C07281=1059.904,-11.969,431.979,171.523,28.026,155.225
C07282=1059.910,-11.719,431.964,171.524,28.029,155.225
C07283=1059.916,-11.470,431.951,171.526,28.031,155.225
C07284=1059.922,-11.220,431.937,171.528,28.033,155.226
C07285=1059.928,-10.971,431.922,171.529,28.035,155.226
C07286=1059.934,-10.722,431.909,171.531,28.038,155.226
C07287=1059.941,-10.472,431.894,171.532,28.040,155.226
C07288=1059.946,-10.222,431.880,171.534,28.042,155.227
C07289=1059.953,-9.972,431.867,171.536,28.045,155.227
C07290=1059.959,-9.723,431.852,171.537,28.047,155.227
C07291=1059.965,-9.473,431.838,171.539,28.049,155.228
C07292=1059.972,-9.225,431.824,171.540,28.051,155.228
C07293=1059.977,-8.975,431.810,171.541,28.054,155.228
C07294=1059.983,-8.725,431.796,171.543,28.056,155.228
C07295=1059.990,-8.476,431.782,171.545,28.058,155.229
C07296=1059.996,-8.226,431.767,171.546,28.060,155.229
C07297=1060.001,-7.977,431.753,171.548,28.063,155.229
C07298=1060.008,-7.727,431.739,171.549,28.065,155.230
C07299=1060.014,-7.478,431.725,171.551,28.067,155.230
C07300=1060.020,-7.228,431.710,171.553,28.069,155.230
C07301=1060.027,-6.979,431.696,171.554,28.072,155.230
C07302=1060.033,-6.729,431.682,171.556,28.074,155.231
C07303=1060.039,-6.480,431.668,171.557,28.076,155.231
C07304=1060.045,-6.229,431.653,171.558,28.079,155.231
C07305=1060.051,-5.981,431.639,171.560,28.081,155.232
C07306=1060.057,-5.731,431.625,171.562,28.083,155.232
C07307=1060.063,-5.482,431.611,171.563,28.085,155.232
C07308=1060.070,-5.232,431.597,171.565,28.088,155.232
C07309=1060.076,-4.983,431.582,171.566,28.090,155.233
C07310=1060.082,-4.732,431.568,171.568,28.092,155.233
C07311=1060.088,-4.484,431.554,171.570,28.094,155.233
C07312=1060.095,-4.234,431.539,171.571,28.097,155.233
C07313=1060.101,-3.984,431.525,171.573,28.099,155.234
C07314=1060.106,-3.735,431.510,171.574,28.101,155.234
C07315=1060.113,-3.485,431.497,171.575,28.104,155.234
C07316=1060.119,-3.236,431.482,171.577,28.106,155.235
C07317=1060.125,-2.986,431.467,171.579,28.108,155.235
C07318=1060.131,-2.737,431.453,171.580,28.110,155.235
C07319=1060.137,-2.455,431.437,171.582,28.113,155.236
C07320=1060.145,-2.174,431.420,171.583,28.116,155.236
C07321=1060.151,-1.893,431.404,171.585,28.118,155.236
C07322=1060.158,-1.612,431.388,171.587,28.121,155.237
C07323=1060.164,-1.362,431.373,171.588,28.123,155.237
C07324=1060.170,-1.113,431.359,171.590,28.126,155.237
C07325=1060.176,-0.863,431.344,171.591,28.128,155.238
C07326=1060.182,-0.614,431.330,171.593,28.131,155.238
C07327=1060.188,-0.364,431.315,171.595,28.134,155.238
C07328=1060.194,-0.114,431.301,171.596,28.136,155.239
C07329=1060.200,0.135,431.286,171.598,28.138,155.239
C07330=1060.207,0.385,431.271,171.600,28.140,155.239
C07331=1060.212,0.634,431.257,171.600,28.143,155.239
C07332=1060.218,0.884,431.242,171.602,28.145,155.240
C07333=1060.224,1.133,431.228,171.603,28.147,155.240
C07334=1060.231,1.383,431.213,171.605,28.150,155.240
C07335=1060.236,1.632,431.198,171.607,28.152,155.241
C07336=1060.243,1.882,431.184,171.608,28.155,155.241
C07337=1060.248,2.131,431.169,171.610,28.157,155.241
C07338=1060.254,2.381,431.154,171.612,28.160,155.242
C07339=1060.260,2.630,431.139,171.612,28.162,155.242
C07340=1060.266,2.879,431.124,171.614,28.164,155.242
C07341=1060.272,3.130,431.110,171.615,28.166,155.242
C07342=1060.278,3.379,431.096,171.617,28.169,155.243
C07343=1060.284,3.628,431.081,171.619,28.171,155.243
C07344=1060.291,3.878,431.066,171.620,28.173,155.243
C07345=1060.297,4.127,431.051,171.622,28.176,155.244
C07346=1060.303,4.377,431.036,171.624,28.179,155.244
C07347=1060.309,4.626,431.021,171.625,28.181,155.244
C07348=1060.315,4.876,431.007,171.626,28.183,155.245
C07349=1060.321,5.125,430.992,171.627,28.186,155.245
C07350=1060.327,5.374,430.978,171.629,28.188,155.245
C07351=1060.333,5.624,430.963,171.631,28.190,155.246
C07352=1060.340,5.874,430.948,171.632,28.193,155.246
C07353=1060.345,6.123,430.933,171.634,28.195,155.246
C07354=1060.352,6.372,430.918,171.636,28.197,155.246
C07355=1060.358,6.622,430.903,171.637,28.200,155.247
C07356=1060.364,6.871,430.889,171.638,28.202,155.247
C07357=1060.370,7.121,430.873,171.640,28.204,155.247
C07358=1060.376,7.371,430.858,171.641,28.207,155.248
C07359=1060.382,7.620,430.844,171.643,28.209,155.248
C07360=1060.388,7.870,430.830,171.644,28.212,155.248
C07361=1060.394,8.119,430.815,171.646,28.214,155.249
C07362=1060.400,8.368,430.800,171.648,28.217,155.249
C07363=1060.406,8.618,430.785,171.648,28.219,155.249
C07364=1060.413,8.868,430.770,171.650,28.221,155.250
C07365=1060.419,9.117,430.755,171.652,28.224,155.250
C07366=1060.425,9.366,430.741,171.653,28.226,155.250
C07367=1060.431,9.616,430.726,171.655,28.228,155.251
C07368=1060.438,9.866,430.711,171.656,28.231,155.251
C07369=1060.444,10.115,430.694,171.658,28.233,155.251
C07370=1060.450,10.364,430.680,171.660,28.236,155.251
C07371=1060.456,10.614,430.665,171.660,28.238,155.252
C07372=1060.462,10.863,430.650,171.662,28.240,155.252
C07373=1060.468,11.112,430.635,171.664,28.243,155.252
C07374=1060.474,11.362,430.620,171.665,28.245,155.253
C07375=1060.481,11.612,430.605,171.667,28.248,155.253
C07376=1060.487,11.861,430.591,171.669,28.250,155.253
C07377=1060.493,12.111,430.575,171.670,28.252,155.254
C07378=1060.499,12.360,430.560,171.671,28.255,155.254
C07379=1060.505,12.610,430.545,171.672,28.257,155.254
C07380=1060.511,12.859,430.531,171.674,28.259,155.255
C07381=1060.518,13.109,430.515,171.676,28.262,155.255
C07382=1060.524,13.357,430.500,171.677,28.264,155.255
C07383=1060.531,13.642,430.483,171.679,28.267,155.256
C07384=1060.538,13.925,430.466,171.681,28.269,155.256
C07385=1060.546,14.208,430.449,171.682,28.272,155.256
C07386=1060.552,14.491,430.432,171.684,28.275,155.257
C07387=1060.559,14.740,430.416,171.685,28.277,155.257
C07388=1060.564,14.990,430.401,171.687,28.280,155.257
C07389=1060.570,15.239,430.386,171.689,28.282,155.258
C07390=1060.576,15.489,430.371,171.690,28.285,155.258
C07391=1060.582,15.739,430.356,171.692,28.287,155.258
C07392=1060.588,15.987,430.340,171.693,28.290,155.259
C07393=1060.595,16.237,430.325,171.694,28.292,155.259
C07394=1060.600,16.487,430.310,171.696,28.295,155.259
C07395=1060.607,16.737,430.295,171.697,28.297,155.260
C07396=1060.613,16.986,430.279,171.699,28.299,155.260
C07397=1060.618,17.235,430.264,171.701,28.302,155.260
C07398=1060.625,17.485,430.249,171.702,28.304,155.261
C07399=1060.631,17.734,430.234,171.703,28.307,155.261
C07400=1060.637,17.984,430.218,171.705,28.309,155.261
C07401=1060.643,18.233,430.203,171.706,28.312,155.262
C07402=1060.648,18.483,430.188,171.708,28.314,155.262
C07403=1060.655,18.732,430.172,171.709,28.317,155.262
C07404=1060.662,18.981,430.157,171.711,28.319,155.263
C07405=1060.667,19.231,430.142,171.713,28.321,155.263
C07406=1060.674,19.480,430.126,171.713,28.324,155.263
C07407=1060.680,19.730,430.111,171.715,28.326,155.264
C07408=1060.685,19.979,430.096,171.716,28.329,155.264
C07409=1060.692,20.228,430.080,171.718,28.331,155.264
C07410=1060.698,20.478,430.065,171.720,28.334,155.265
C07411=1060.704,20.728,430.050,171.721,28.336,155.265
C07412=1060.710,20.977,430.033,171.722,28.339,155.265
C07413=1060.716,21.227,430.019,171.724,28.341,155.266
C07414=1060.722,21.476,430.002,171.725,28.344,155.266
C07415=1060.728,21.725,429.988,171.727,28.346,155.266
C07416=1060.734,21.974,429.971,171.728,28.349,155.267
C07417=1060.740,22.224,429.956,171.730,28.351,155.267
C07418=1060.746,22.474,429.941,171.732,28.354,155.267
C07419=1060.753,22.723,429.925,171.732,28.356,155.268
C07420=1060.758,22.973,429.910,171.734,28.359,155.268
C07421=1060.765,23.222,429.894,171.736,28.361,155.268
C07422=1060.770,23.471,429.879,171.737,28.364,155.269
C07423=1060.777,23.720,429.863,171.739,28.366,155.269
C07424=1060.782,23.970,429.848,171.741,28.369,155.269
C07425=1060.789,24.219,429.832,171.741,28.371,155.270
C07426=1060.795,24.469,429.816,171.743,28.374,155.270
C07427=1060.801,24.718,429.801,171.744,28.376,155.270
C07428=1060.807,24.968,429.785,171.746,28.379,155.271
C07429=1060.814,25.217,429.770,171.748,28.381,155.271
C07430=1060.819,25.467,429.754,171.749,28.384,155.271
C07431=1060.825,25.717,429.738,171.750,28.386,155.272
C07432=1060.831,25.966,429.723,171.752,28.388,155.272
C07433=1060.837,26.215,429.707,171.753,28.391,155.272
C07434=1060.844,26.465,429.692,171.755,28.393,155.273
C07435=1060.849,26.714,429.676,171.756,28.396,155.273
C07436=1060.856,26.963,429.660,171.758,28.398,155.273
C07437=1060.862,27.213,429.645,171.759,28.400,155.274
C07438=1060.868,27.462,429.628,171.760,28.403,155.274
C07439=1060.874,27.712,429.613,171.762,28.406,155.275
C07440=1060.880,27.961,429.597,171.764,28.408,155.275
C07441=1060.887,28.210,429.581,171.765,28.411,155.275
C07442=1060.892,28.460,429.566,171.767,28.413,155.275
C07443=1060.898,28.710,429.550,171.768,28.416,155.276
C07444=1060.905,28.959,429.534,171.769,28.418,155.276
C07445=1060.911,29.209,429.518,171.771,28.421,155.277
C07446=1060.917,29.458,429.502,171.772,28.423,155.277
C07447=1060.924,29.743,429.485,171.774,28.426,155.277
C07448=1060.930,30.027,429.466,171.776,28.429,155.278
C07449=1060.938,30.312,429.449,171.777,28.432,155.278
C07450=1060.944,30.596,429.430,171.779,28.435,155.279
C07451=1060.950,30.846,429.414,171.780,28.438,155.279
C07452=1060.956,31.096,429.398,171.782,28.440,155.279
C07453=1060.962,31.345,429.383,171.784,28.443,155.280
C07454=1060.968,31.594,429.366,171.785,28.445,155.280
C07455=1060.974,31.844,429.351,171.786,28.447,155.280
C07456=1060.980,32.093,429.334,171.787,28.450,155.281
C07457=1060.987,32.342,429.319,171.789,28.452,155.281
C07458=1060.993,32.592,429.303,171.791,28.455,155.281
C07459=1060.998,32.842,429.287,171.792,28.458,155.282
C07460=1061.004,33.091,429.271,171.794,28.460,155.282
C07461=1061.011,33.340,429.255,171.795,28.463,155.282
C07462=1061.017,33.589,429.239,171.796,28.465,155.283
C07463=1061.023,33.839,429.223,171.798,28.468,155.283
C07464=1061.028,34.089,429.207,171.799,28.470,155.283
C07465=1061.035,34.338,429.191,171.801,28.473,155.284
C07466=1061.041,34.587,429.175,171.803,28.476,155.284
C07467=1061.047,34.836,429.159,171.803,28.478,155.284
C07468=1061.053,35.086,429.143,171.805,28.480,155.285
C07469=1061.059,35.335,429.126,171.807,28.483,155.285
C07470=1061.065,35.585,429.111,171.808,28.485,155.286
C07471=1061.071,35.834,429.095,171.810,28.488,155.286
C07472=1061.077,36.083,429.079,171.812,28.490,155.286
C07473=1061.083,36.333,429.063,171.812,28.493,155.287
C07474=1061.089,36.582,429.046,171.814,28.495,155.287
C07475=1061.096,36.831,429.031,171.815,28.498,155.287
C07476=1061.102,37.081,429.014,171.817,28.501,155.288
C07477=1061.108,37.331,428.998,171.819,28.503,155.288
C07478=1061.114,37.580,428.982,171.820,28.506,155.288
C07479=1061.120,37.829,428.965,171.821,28.508,155.289
C07480=1061.126,38.079,428.950,171.823,28.511,155.289
C07481=1061.132,38.329,428.934,171.824,28.513,155.289
C07482=1061.138,38.578,428.917,171.826,28.516,155.290
C07483=1061.144,38.827,428.901,171.827,28.518,155.290
C07484=1061.150,39.077,428.885,171.828,28.521,155.291
C07485=1061.156,39.326,428.868,171.830,28.523,155.291
C07486=1061.162,39.575,428.852,171.831,28.526,155.291
C07487=1061.168,39.825,428.836,171.833,28.529,155.292
C07488=1061.173,40.074,428.820,171.835,28.532,155.292
C07489=1061.179,40.323,428.803,171.836,28.534,155.292
C07490=1061.185,40.573,428.787,171.837,28.536,155.293
C07491=1061.192,40.823,428.771,171.838,28.539,155.293
C07492=1061.198,41.072,428.754,171.840,28.541,155.293
C07493=1061.204,41.321,428.737,171.842,28.544,155.294
C07494=1061.210,41.570,428.721,171.843,28.547,155.294
C07495=1061.216,41.820,428.705,171.844,28.549,155.294
C07496=1061.222,42.069,428.689,171.846,28.552,155.295
C07497=1061.228,42.318,428.672,171.847,28.555,155.295
C07498=1061.234,42.568,428.656,171.849,28.557,155.296
C07499=1061.240,42.817,428.640,171.851,28.560,155.296
C07500=1061.246,43.067,428.623,171.852,28.562,155.296
C07501=1061.252,43.316,428.607,171.853,28.564,155.297
C07502=1061.258,43.566,428.591,171.854,28.567,155.297
C07503=1061.264,43.815,428.574,171.856,28.570,155.297
C07504=1061.270,44.064,428.557,171.858,28.573,155.298
C07505=1061.276,44.313,428.541,171.859,28.575,155.298
C07506=1061.282,44.563,428.524,171.860,28.577,155.299
C07507=1061.288,44.812,428.508,171.862,28.580,155.299
C07508=1061.294,45.062,428.491,171.863,28.583,155.299
C07509=1061.300,45.312,428.475,171.865,28.586,155.300
C07510=1061.306,45.561,428.458,171.866,28.588,155.300
C07511=1061.312,45.845,428.439,171.868,28.591,155.300
C07512=1061.319,46.130,428.420,171.870,28.594,155.301
C07513=1061.326,46.414,428.401,171.871,28.597,155.301
C07514=1061.333,46.699,428.382,171.873,28.600,155.302
C07515=1061.339,46.948,428.366,171.874,28.603,155.302
C07516=1061.344,47.198,428.349,171.876,28.605,155.302
C07517=1061.350,47.447,428.332,171.877,28.608,155.303
C07518=1061.356,47.696,428.316,171.878,28.611,155.303
C07519=1061.362,47.946,428.299,171.880,28.613,155.304
C07520=1061.368,48.196,428.283,171.881,28.616,155.304
C07521=1061.374,48.444,428.266,171.883,28.618,155.304
C07522=1061.380,48.694,428.249,171.885,28.621,155.305
C07523=1061.385,48.943,428.233,171.885,28.624,155.305
C07524=1061.392,49.192,428.216,171.887,28.627,155.306
C07525=1061.398,49.442,428.199,171.889,28.629,155.306
C07526=1061.404,49.691,428.183,171.890,28.632,155.306
C07527=1061.410,49.940,428.165,171.892,28.634,155.307
C07528=1061.416,50.190,428.149,171.892,28.637,155.307
C07529=1061.422,50.439,428.133,171.894,28.639,155.307
C07530=1061.428,50.689,428.115,171.896,28.642,155.308
C07531=1061.434,50.938,428.098,171.897,28.645,155.308
C07532=1061.440,51.188,428.082,171.899,28.647,155.309
C07533=1061.445,51.437,428.065,171.900,28.650,155.309
C07534=1061.452,51.687,428.048,171.901,28.652,155.309
C07535=1061.458,51.935,428.031,171.903,28.655,155.310
C07536=1061.464,52.185,428.015,171.905,28.658,155.310
C07537=1061.469,52.434,427.998,171.906,28.661,155.310
C07538=1061.475,52.683,427.981,171.908,28.663,155.311
C07539=1061.482,52.933,427.964,171.908,28.665,155.311
C07540=1061.487,53.182,427.947,171.910,28.668,155.311
C07541=1061.493,53.432,427.930,171.912,28.671,155.312
C07542=1061.500,53.681,427.913,171.913,28.673,155.312
C07543=1061.505,53.931,427.896,171.915,28.676,155.313
C07544=1061.512,54.179,427.879,171.916,28.678,155.313
C07545=1061.518,54.429,427.863,171.917,28.681,155.313
C07546=1061.523,54.679,427.846,171.919,28.683,155.314
C07547=1061.530,54.928,427.829,171.921,28.686,155.314
C07548=1061.536,55.177,427.813,171.922,28.689,155.314
C07549=1061.542,55.427,427.795,171.924,28.692,155.315
C07550=1061.548,55.676,427.778,171.924,28.694,155.315
C07551=1061.554,55.925,427.761,171.926,28.697,155.316
C07552=1061.560,56.174,427.744,171.928,28.699,155.316
C07553=1061.566,56.424,427.727,171.929,28.702,155.316
C07554=1061.572,56.673,427.710,171.931,28.704,155.317
C07555=1061.578,56.923,427.693,171.932,28.707,155.317
C07556=1061.584,57.172,427.676,171.933,28.710,155.317
C07557=1061.590,57.421,427.660,171.935,28.712,155.318
C07558=1061.596,57.670,427.642,171.937,28.715,155.318
C07559=1061.602,57.920,427.626,171.938,28.717,155.319
C07560=1061.608,58.169,427.608,171.940,28.720,155.319
C07561=1061.614,58.418,427.591,171.940,28.723,155.319
C07562=1061.621,58.668,427.574,171.942,28.725,155.320
C07563=1061.626,58.917,427.557,171.944,28.728,155.320
C07564=1061.633,59.167,427.540,171.945,28.730,155.320
C07565=1061.639,59.416,427.523,171.947,28.733,155.321
C07566=1061.645,59.665,427.506,171.948,28.735,155.321
C07567=1061.651,59.915,427.489,171.949,28.738,155.322
C07568=1061.657,60.164,427.472,171.951,28.741,155.322
C07569=1061.664,60.414,427.454,171.953,28.743,155.322
C07570=1061.669,60.663,427.438,171.954,28.746,155.323
C07571=1061.675,60.912,427.420,171.956,28.748,155.323
C07572=1061.682,61.161,427.403,171.957,28.750,155.323
C07573=1061.688,61.411,427.387,171.958,28.753,155.324
C07574=1061.694,61.660,427.369,171.960,28.756,155.324
C07575=1061.701,61.944,427.350,171.961,28.759,155.324
C07576=1061.708,62.228,427.330,171.963,28.762,155.325
C07577=1061.715,62.514,427.310,171.965,28.765,155.325
C07578=1061.721,62.797,427.291,171.966,28.768,155.326
C07579=1061.728,63.047,427.274,171.968,28.770,155.326
C07580=1061.734,63.296,427.256,171.970,28.773,155.326
C07581=1061.740,63.546,427.239,171.971,28.775,155.327
C07582=1061.747,63.794,427.222,171.973,28.778,155.327
C07583=1061.753,64.044,427.204,171.974,28.780,155.328
C07584=1061.759,64.293,427.188,171.975,28.783,155.328
C07585=1061.765,64.543,427.170,171.977,28.786,155.328
C07586=1061.770,64.792,427.153,171.978,28.788,155.329
C07587=1061.776,65.041,427.136,171.980,28.791,155.329
C07588=1061.783,65.291,427.118,171.982,28.793,155.329
C07589=1061.789,65.539,427.101,171.982,28.796,155.330
C07590=1061.795,65.789,427.083,171.984,28.799,155.330
C07591=1061.800,66.039,427.066,171.986,28.802,155.331
C07592=1061.807,66.288,427.049,171.987,28.804,155.331
C07593=1061.813,66.537,427.031,171.989,28.806,155.331
C07594=1061.818,66.786,427.014,171.991,28.809,155.332
C07595=1061.825,67.036,426.996,171.991,28.812,155.332
C07596=1061.830,67.285,426.979,171.993,28.815,155.333
C07597=1061.837,67.535,426.961,171.994,28.817,155.333
C07598=1061.843,67.783,426.944,171.996,28.820,155.333
C07599=1061.849,68.033,426.926,171.998,28.822,155.334
C07600=1061.854,68.283,426.909,171.999,28.825,155.334
C07601=1061.860,68.532,426.891,172.000,28.828,155.334
C07602=1061.867,68.781,426.874,172.002,28.830,155.335
C07603=1061.873,69.031,426.856,172.003,28.833,155.335
C07604=1061.878,69.280,426.839,172.005,28.835,155.336
C07605=1061.885,69.529,426.821,172.007,28.838,155.336
C07606=1061.891,69.778,426.804,172.007,28.841,155.336
C07607=1061.897,70.028,426.786,172.009,28.843,155.337
C07608=1061.902,70.277,426.768,172.010,28.846,155.337
C07609=1061.908,70.526,426.751,172.012,28.848,155.337
C07610=1061.915,70.776,426.733,172.014,28.851,155.338
C07611=1061.920,71.025,426.716,172.015,28.854,155.338
C07612=1061.926,71.274,426.698,172.016,28.856,155.339
C07613=1061.932,71.523,426.680,172.018,28.859,155.339
C07614=1061.938,71.773,426.662,172.019,28.862,155.339
C07615=1061.944,72.022,426.645,172.021,28.865,155.340
C07616=1061.950,72.272,426.627,172.023,28.867,155.340
C07617=1061.956,72.520,426.609,172.024,28.870,155.341
C07618=1061.962,72.770,426.591,172.025,28.872,155.341
C07619=1061.968,73.019,426.574,172.027,28.875,155.341
C07620=1061.974,73.269,426.556,172.028,28.878,155.342
C07621=1061.979,73.518,426.538,172.030,28.881,155.342
C07622=1061.986,73.767,426.521,172.031,28.883,155.343
C07623=1061.992,74.016,426.503,172.032,28.886,155.343
C07624=1061.998,74.266,426.485,172.034,28.888,155.343
C07625=1062.004,74.516,426.467,172.035,28.891,155.344
C07626=1062.010,74.764,426.449,172.037,28.894,155.344
C07627=1062.016,75.014,426.431,172.039,28.896,155.344
C07628=1062.021,75.263,426.414,172.040,28.899,155.345
C07629=1062.028,75.513,426.396,172.041,28.902,155.345
C07630=1062.034,75.761,426.379,172.043,28.904,155.346
C07631=1062.040,76.011,426.361,172.044,28.907,155.346
C07632=1062.046,76.259,426.342,172.046,28.909,155.346
C07633=1062.052,76.509,426.324,172.048,28.912,155.347
C07634=1062.058,76.759,426.307,172.049,28.915,155.347
C07635=1062.064,77.008,426.289,172.050,28.917,155.348
C07636=1062.070,77.258,426.271,172.052,28.920,155.348
C07637=1062.075,77.506,426.253,172.053,28.922,155.348
C07638=1062.082,77.756,426.235,172.055,28.925,155.349
C07639=1062.088,78.040,426.215,172.056,28.928,155.349
C07640=1062.096,78.324,426.194,172.058,28.931,155.350
C07641=1062.102,78.608,426.174,172.060,28.934,155.350
C07642=1062.109,78.892,426.153,172.061,28.937,155.351
C07643=1062.115,79.142,426.135,172.063,28.940,155.351
C07644=1062.121,79.391,426.118,172.065,28.943,155.351
C07645=1062.126,79.641,426.099,172.066,28.946,155.352
C07646=1062.132,79.890,426.080,172.068,28.948,155.352
C07647=1062.138,80.139,426.063,172.068,28.951,155.353
C07648=1062.144,80.389,426.045,172.070,28.953,155.353
C07649=1062.150,80.637,426.027,172.072,28.956,155.353
C07650=1062.156,80.887,426.009,172.073,28.959,155.354
C07651=1062.162,81.135,425.990,172.075,28.961,155.354
C07652=1062.168,81.385,425.973,172.077,28.964,155.354
C07653=1062.173,81.635,425.954,172.077,28.967,155.355
C07654=1062.179,81.884,425.936,172.079,28.969,155.355
C07655=1062.185,82.133,425.918,172.081,28.972,155.356
C07656=1062.191,82.383,425.900,172.082,28.975,155.356
C07657=1062.197,82.631,425.882,172.084,28.978,155.356
C07658=1062.203,82.881,425.864,172.086,28.980,155.357
C07659=1062.209,83.130,425.845,172.086,28.983,155.357
C07660=1062.215,83.380,425.827,172.088,28.985,155.358
C07661=1062.221,83.629,425.808,172.090,28.988,155.358
C07662=1062.227,83.878,425.791,172.091,28.991,155.358
C07663=1062.233,84.128,425.773,172.093,28.993,155.359
C07664=1062.239,84.377,425.754,172.095,28.996,155.359
C07665=1062.245,84.626,425.736,172.095,28.999,155.360
C07666=1062.250,84.875,425.717,172.097,29.001,155.360
C07667=1062.256,85.125,425.699,172.098,29.004,155.360
C07668=1062.262,85.373,425.681,172.100,29.007,155.361
C07669=1062.268,85.623,425.663,172.102,29.009,155.361
C07670=1062.275,85.872,425.644,172.103,29.012,155.361
C07671=1062.280,86.121,425.627,172.105,29.015,155.362
C07672=1062.286,86.371,425.608,172.106,29.017,155.362
C07673=1062.292,86.620,425.590,172.107,29.020,155.363
C07674=1062.299,86.870,425.571,172.109,29.023,155.363
C07675=1062.304,87.118,425.553,172.111,29.025,155.364
C07676=1062.310,87.368,425.535,172.112,29.028,155.364
C07677=1062.317,87.617,425.516,172.114,29.030,155.364
C07678=1062.322,87.866,425.498,172.116,29.033,155.365
C07679=1062.328,88.115,425.479,172.116,29.036,155.365
C07680=1062.334,88.365,425.461,172.118,29.038,155.365
C07681=1062.341,88.614,425.443,172.120,29.041,155.366
C07682=1062.346,88.863,425.425,172.121,29.044,155.366
C07683=1062.352,89.113,425.406,172.123,29.047,155.367
C07684=1062.358,89.362,425.387,172.125,29.049,155.367
C07685=1062.365,89.611,425.369,172.125,29.051,155.367
C07686=1062.370,89.860,425.351,172.127,29.054,155.368
C07687=1062.376,90.109,425.332,172.129,29.057,155.368
C07688=1062.382,90.358,425.313,172.130,29.060,155.369
C07689=1062.388,90.608,425.295,172.132,29.062,155.369
C07690=1062.394,90.857,425.277,172.134,29.065,155.369
C07691=1062.400,91.106,425.258,172.135,29.068,155.370
C07692=1062.406,91.356,425.240,172.136,29.070,155.370
C07693=1062.412,91.605,425.221,172.138,29.073,155.371
C07694=1062.418,91.854,425.202,172.139,29.076,155.371
C07695=1062.424,92.103,425.184,172.141,29.078,155.371
C07696=1062.429,92.353,425.165,172.143,29.081,155.372
C07697=1062.436,92.602,425.146,172.144,29.084,155.372
C07698=1062.441,92.851,425.128,172.146,29.086,155.372
C07699=1062.447,93.100,425.110,172.147,29.089,155.373
C07700=1062.453,93.350,425.090,172.148,29.092,155.373
C07701=1062.459,93.599,425.072,172.150,29.094,155.374
C07702=1062.464,93.848,425.053,172.151,29.097,155.374
C07703=1062.471,94.132,425.032,172.153,29.100,155.375
C07704=1062.479,94.416,425.011,172.155,29.103,155.375
C07705=1062.485,94.701,424.989,172.156,29.107,155.376
C07706=1062.492,94.985,424.968,172.158,29.109,155.376
C07707=1062.498,95.234,424.949,172.160,29.112,155.376
C07708=1062.504,95.482,424.930,172.161,29.115,155.377
C07709=1062.509,95.732,424.912,172.163,29.117,155.377
C07710=1062.515,95.982,424.893,172.164,29.120,155.378
C07711=1062.521,96.231,424.874,172.166,29.123,155.378
C07712=1062.527,96.480,424.855,172.168,29.126,155.378
C07713=1062.533,96.729,424.836,172.169,29.128,155.379
C07714=1062.539,96.978,424.818,172.170,29.131,155.379
C07715=1062.545,97.227,424.799,172.172,29.133,155.379
C07716=1062.551,97.477,424.780,172.174,29.136,155.380
C07717=1062.557,97.726,424.761,172.175,29.139,155.380
C07718=1062.563,97.976,424.743,172.177,29.141,155.381
C07719=1062.569,98.225,424.723,172.178,29.144,155.381
C07720=1062.574,98.474,424.705,172.180,29.147,155.381
C07721=1062.580,98.723,424.686,172.182,29.150,155.382
C07722=1062.587,98.972,424.667,172.182,29.152,155.382
C07723=1062.592,99.222,424.648,172.184,29.155,155.383
C07724=1062.599,99.471,424.629,172.186,29.158,155.383
C07725=1062.604,99.720,424.610,172.187,29.160,155.384
C07726=1062.611,99.969,424.592,172.189,29.163,155.384
C07727=1062.616,100.219,424.572,172.191,29.165,155.384
C07728=1062.622,100.467,424.554,172.192,29.168,155.385
C07729=1062.628,100.717,424.535,172.194,29.171,155.385
C07730=1062.634,100.966,424.516,172.195,29.173,155.385
C07731=1062.640,101.215,424.497,172.196,29.176,155.386
C07732=1062.646,101.465,424.478,172.198,29.179,155.386
C07733=1062.652,101.714,424.459,172.200,29.182,155.387
C07734=1062.658,101.963,424.440,172.201,29.184,155.387
C07735=1062.664,102.213,424.420,172.203,29.187,155.387
C07736=1062.669,102.461,424.401,172.205,29.190,155.388
C07737=1062.675,102.710,424.382,172.206,29.192,155.388
C07738=1062.681,102.959,424.363,172.207,29.195,155.389
C07739=1062.687,103.209,424.344,172.209,29.198,155.389
C07740=1062.692,103.458,424.324,172.210,29.200,155.390
C07741=1062.699,103.707,424.306,172.212,29.203,155.390
C07742=1062.705,103.957,424.287,172.214,29.206,155.390
C07743=1062.710,104.206,424.267,172.215,29.209,155.391
C07744=1062.716,104.455,424.247,172.217,29.211,155.391
C07745=1062.723,104.704,424.229,172.219,29.214,155.392
C07746=1062.728,104.953,424.210,172.220,29.217,155.392
C07747=1062.733,105.202,424.191,172.221,29.219,155.392
C07748=1062.739,105.452,424.171,172.223,29.222,155.393
C07749=1062.746,105.701,424.153,172.224,29.225,155.393
C07750=1062.752,105.949,424.133,172.226,29.228,155.394
C07751=1062.757,106.199,424.114,172.228,29.230,155.394
C07752=1062.763,106.448,424.094,172.229,29.233,155.394
C07753=1062.769,106.697,424.076,172.231,29.235,155.395
C07754=1062.775,106.946,424.056,172.233,29.238,155.395
C07755=1062.781,107.196,424.036,172.234,29.241,155.395
C07756=1062.787,107.445,424.017,172.235,29.243,155.396
C07757=1062.792,107.695,423.998,172.237,29.246,155.396
C07758=1062.799,107.943,423.979,172.238,29.249,155.397
C07759=1062.805,108.193,423.959,172.240,29.251,155.397
C07760=1062.811,108.442,423.940,172.242,29.254,155.398
C07761=1062.816,108.691,423.921,172.243,29.257,155.398
C07762=1062.823,108.940,423.901,172.245,29.260,155.398
C07763=1062.829,109.189,423.882,172.247,29.262,155.399
C07764=1062.834,109.439,423.863,172.248,29.265,155.399
C07765=1062.840,109.688,423.843,172.250,29.268,155.400
C07766=1062.846,109.937,423.824,172.251,29.270,155.400
C07767=1062.853,110.221,423.801,172.253,29.273,155.400
C07768=1062.860,110.505,423.780,172.255,29.277,155.401
C07769=1062.867,110.789,423.758,172.257,29.279,155.401
C07770=1062.874,111.074,423.736,172.258,29.283,155.402
C07771=1062.879,111.323,423.716,172.260,29.285,155.402
C07772=1062.885,111.572,423.697,172.262,29.288,155.402
C07773=1062.891,111.821,423.677,172.263,29.290,155.403
C07774=1062.897,112.070,423.657,172.265,29.293,155.403
C07775=1062.903,112.319,423.637,172.267,29.296,155.404
C07776=1062.909,112.569,423.618,172.268,29.298,155.404
C07777=1062.914,112.818,423.599,172.270,29.301,155.405
C07778=1062.920,113.067,423.579,172.272,29.304,155.405
C07779=1062.926,113.316,423.560,172.272,29.306,155.405
C07780=1062.932,113.565,423.540,172.274,29.309,155.406
C07781=1062.938,113.814,423.521,172.276,29.312,155.406
C07782=1062.944,114.063,423.501,172.277,29.315,155.407
C07783=1062.949,114.313,423.481,172.279,29.317,155.407
C07784=1062.955,114.562,423.461,172.281,29.320,155.407
C07785=1062.961,114.811,423.442,172.282,29.323,155.408
C07786=1062.967,115.060,423.422,172.284,29.326,155.408
C07787=1062.973,115.309,423.403,172.286,29.329,155.409
C07788=1062.979,115.558,423.383,172.287,29.332,155.409
C07789=1062.984,115.808,423.363,172.289,29.334,155.410
C07790=1062.990,116.057,423.343,172.291,29.337,155.410
C07791=1062.996,116.306,423.323,172.291,29.340,155.410
C07792=1063.001,116.555,423.304,172.293,29.342,155.411
C07793=1063.007,116.804,423.284,172.295,29.345,155.411
C07794=1063.013,117.053,423.265,172.296,29.348,155.412
C07795=1063.018,117.302,423.244,172.298,29.350,155.412
C07796=1063.024,117.551,423.224,172.300,29.353,155.412
C07797=1063.030,117.801,423.205,172.301,29.356,155.413
C07798=1063.036,118.050,423.185,172.303,29.359,155.413
C07799=1063.042,118.299,423.165,172.305,29.361,155.414
C07800=1063.047,118.549,423.145,172.306,29.364,155.414
C07801=1063.053,118.797,423.125,172.308,29.367,155.414
C07802=1063.059,119.046,423.105,172.310,29.370,155.415
C07803=1063.065,119.296,423.086,172.311,29.373,155.415
C07804=1063.071,119.545,423.066,172.312,29.375,155.416
C07805=1063.076,119.794,423.045,172.314,29.378,155.416
C07806=1063.082,120.043,423.026,172.315,29.381,155.417
C07807=1063.088,120.292,423.006,172.317,29.384,155.417
C07808=1063.095,120.541,422.986,172.319,29.386,155.417
C07809=1063.100,120.791,422.965,172.320,29.389,155.418
C07810=1063.106,121.040,422.946,172.322,29.392,155.418
C07811=1063.112,121.289,422.926,172.324,29.394,155.419
C07812=1063.118,121.538,422.906,172.325,29.397,155.419
C07813=1063.123,121.787,422.885,172.327,29.400,155.419
C07814=1063.128,122.036,422.866,172.329,29.403,155.420
C07815=1063.135,122.286,422.846,172.330,29.405,155.420
C07816=1063.141,122.534,422.826,172.332,29.408,155.421
C07817=1063.147,122.783,422.806,172.334,29.411,155.421
C07818=1063.152,123.032,422.785,172.335,29.413,155.421
C07819=1063.158,123.282,422.766,172.337,29.416,155.422
C07820=1063.164,123.531,422.746,172.339,29.419,155.422
C07821=1063.171,123.780,422.726,172.340,29.422,155.423
C07822=1063.176,124.029,422.705,172.342,29.424,155.423
C07823=1063.182,124.278,422.685,172.344,29.427,155.423
C07824=1063.188,124.527,422.665,172.344,29.430,155.424
C07825=1063.193,124.777,422.646,172.346,29.432,155.424
C07826=1063.199,125.026,422.625,172.348,29.435,155.425
C07827=1063.205,125.275,422.605,172.350,29.438,155.425
C07828=1063.211,125.524,422.585,172.351,29.440,155.426
C07829=1063.217,125.773,422.565,172.353,29.443,155.426
C07830=1063.223,126.022,422.545,172.355,29.446,155.426
C07831=1063.230,126.306,422.522,172.357,29.449,155.427
C07832=1063.237,126.590,422.498,172.359,29.452,155.427
C07833=1063.244,126.875,422.475,172.360,29.455,155.428
C07834=1063.249,127.158,422.452,172.362,29.458,155.428
C07835=1063.255,127.407,422.433,172.364,29.461,155.429
C07836=1063.262,127.657,422.412,172.365,29.464,155.429
C07837=1063.268,127.906,422.392,172.367,29.466,155.429
C07838=1063.273,128.155,422.372,172.369,29.469,155.430
C07839=1063.280,128.404,422.351,172.371,29.472,155.430
C07840=1063.286,128.653,422.331,172.372,29.474,155.431
C07841=1063.291,128.902,422.311,172.374,29.477,155.431
C07842=1063.297,129.151,422.291,172.376,29.480,155.431
C07843=1063.304,129.401,422.271,172.377,29.483,155.432
C07844=1063.309,129.650,422.250,172.379,29.485,155.432
C07845=1063.315,129.898,422.230,172.381,29.487,155.433
C07846=1063.322,130.148,422.210,172.382,29.490,155.433
C07847=1063.327,130.397,422.189,172.384,29.493,155.433
C07848=1063.333,130.646,422.169,172.386,29.496,155.434
C07849=1063.339,130.895,422.149,172.387,29.498,155.434
C07850=1063.345,131.144,422.128,172.389,29.501,155.435
C07851=1063.351,131.393,422.108,172.391,29.504,155.435
C07852=1063.358,131.642,422.087,172.392,29.506,155.435
C07853=1063.363,131.891,422.067,172.394,29.509,155.436
C07854=1063.369,132.140,422.047,172.396,29.512,155.436
C07855=1063.375,132.390,422.026,172.397,29.515,155.437
C07856=1063.381,132.639,422.006,172.399,29.517,155.437
C07857=1063.386,132.888,421.985,172.401,29.520,155.437
C07858=1063.392,133.136,421.965,172.403,29.523,155.438
C07859=1063.398,133.386,421.944,172.404,29.525,155.438
C07860=1063.403,133.635,421.923,172.406,29.528,155.439
C07861=1063.409,133.884,421.903,172.408,29.531,155.439
C07862=1063.415,134.134,421.882,172.409,29.534,155.440
C07863=1063.421,134.382,421.862,172.411,29.537,155.440
C07864=1063.427,134.631,421.841,172.413,29.540,155.440
C07865=1063.433,134.881,421.820,172.414,29.542,155.441
C07866=1063.439,135.130,421.800,172.416,29.545,155.441
C07867=1063.444,135.378,421.779,172.418,29.548,155.442
C07868=1063.451,135.628,421.759,172.419,29.550,155.442
C07869=1063.456,135.877,421.738,172.421,29.553,155.442
C07870=1063.462,136.125,421.717,172.423,29.556,155.443
C07871=1063.468,136.375,421.697,172.424,29.559,155.443
C07872=1063.473,136.624,421.676,172.426,29.561,155.444
C07873=1063.480,136.874,421.656,172.428,29.564,155.444
C07874=1063.486,137.122,421.634,172.429,29.567,155.444
C07875=1063.491,137.371,421.614,172.431,29.569,155.445
C07876=1063.498,137.620,421.593,172.433,29.572,155.445
C07877=1063.503,137.869,421.572,172.435,29.575,155.446
C07878=1063.508,138.118,421.552,172.436,29.577,155.446
C07879=1063.515,138.367,421.531,172.438,29.580,155.447
C07880=1063.520,138.616,421.510,172.440,29.583,155.447
C07881=1063.526,138.866,421.489,172.441,29.586,155.447
C07882=1063.532,139.115,421.468,172.443,29.589,155.448
C07883=1063.538,139.363,421.448,172.446,29.592,155.448
C07884=1063.544,139.613,421.426,172.447,29.594,155.449
C07885=1063.549,139.862,421.406,172.449,29.597,155.449
C07886=1063.556,140.111,421.385,172.451,29.600,155.449
C07887=1063.561,140.360,421.364,172.452,29.603,155.450
C07888=1063.567,140.610,421.343,172.454,29.605,155.450
C07889=1063.573,140.858,421.322,172.456,29.608,155.451
C07890=1063.578,141.107,421.301,172.457,29.611,155.451
C07891=1063.585,141.356,421.280,172.459,29.613,155.452
C07892=1063.590,141.605,421.260,172.461,29.616,155.452
C07893=1063.596,141.854,421.238,172.462,29.619,155.452
C07894=1063.602,142.104,421.218,172.464,29.622,155.453
C07895=1063.608,142.388,421.194,172.466,29.625,155.453
C07896=1063.615,142.672,421.170,172.468,29.628,155.454
C07897=1063.622,142.956,421.146,172.470,29.632,155.454
C07898=1063.628,143.239,421.122,172.472,29.634,155.455
C07899=1063.634,143.488,421.100,172.473,29.637,155.455
C07900=1063.640,143.737,421.079,172.475,29.640,155.456
C07901=1063.645,143.987,421.058,172.477,29.643,155.456
C07902=1063.651,144.235,421.037,172.479,29.646,155.456
C07903=1063.658,144.485,421.017,172.481,29.649,155.457
C07904=1063.663,144.733,420.995,172.483,29.651,155.457
C07905=1063.669,144.982,420.974,172.485,29.654,155.458
C07906=1063.675,145.231,420.953,172.486,29.657,155.458
C07907=1063.681,145.481,420.931,172.488,29.659,155.458
C07908=1063.686,145.730,420.911,172.490,29.662,155.459
C07909=1063.692,145.979,420.889,172.491,29.665,155.459
C07910=1063.698,146.228,420.868,172.493,29.667,155.460
C07911=1063.705,146.476,420.847,172.495,29.671,155.460
C07912=1063.710,146.726,420.826,172.496,29.673,155.461
C07913=1063.716,146.975,420.805,172.498,29.676,155.461
C07914=1063.722,147.223,420.783,172.500,29.679,155.461
C07915=1063.728,147.473,420.763,172.502,29.681,155.462
C07916=1063.733,147.722,420.741,172.504,29.684,155.462
C07917=1063.739,147.971,420.720,172.506,29.687,155.463
C07918=1063.745,148.220,420.698,172.508,29.690,155.463
C07919=1063.751,148.469,420.677,172.509,29.692,155.463
C07920=1063.757,148.718,420.656,172.511,29.695,155.464
C07921=1063.762,148.967,420.635,172.513,29.698,155.464
C07922=1063.769,149.216,420.613,172.514,29.701,155.465
C07923=1063.774,149.465,420.592,172.516,29.704,155.465
C07924=1063.780,149.714,420.571,172.518,29.707,155.466
C07925=1063.786,149.963,420.549,172.519,29.709,155.466
C07926=1063.792,150.212,420.528,172.521,29.712,155.466
C07927=1063.797,150.461,420.507,172.523,29.715,155.467
C07928=1063.803,150.710,420.485,172.526,29.718,155.467
C07929=1063.808,150.959,420.464,172.527,29.721,155.468
C07930=1063.814,151.208,420.442,172.529,29.723,155.468
C07931=1063.820,151.458,420.421,172.531,29.726,155.469
C07932=1063.826,151.706,420.399,172.532,29.729,155.469
C07933=1063.832,151.955,420.378,172.534,29.732,155.469
C07934=1063.838,152.204,420.356,172.536,29.734,155.470
C07935=1063.844,152.453,420.335,172.537,29.738,155.470
C07936=1063.849,152.702,420.313,172.539,29.740,155.471
C07937=1063.855,152.951,420.291,172.541,29.743,155.471
C07938=1063.861,153.200,420.270,172.543,29.746,155.472
C07939=1063.866,153.449,420.248,172.545,29.748,155.472
C07940=1063.873,153.698,420.227,172.547,29.751,155.472
C07941=1063.879,153.947,420.205,172.549,29.754,155.473
C07942=1063.884,154.196,420.184,172.550,29.757,155.473
C07943=1063.890,154.445,420.162,172.552,29.760,155.474
C07944=1063.895,154.694,420.140,172.554,29.762,155.474
C07945=1063.901,154.943,420.119,172.555,29.765,155.475
C07946=1063.908,155.192,420.097,172.558,29.768,155.475
C07947=1063.913,155.441,420.076,172.560,29.771,155.475
C07948=1063.919,155.690,420.054,172.561,29.774,155.476
C07949=1063.925,155.939,420.032,172.563,29.777,155.476
C07950=1063.930,156.188,420.011,172.565,29.779,155.477
C07951=1063.936,156.437,419.989,172.566,29.782,155.477
C07952=1063.943,156.686,419.967,172.568,29.785,155.478
C07953=1063.947,156.935,419.945,172.570,29.787,155.478
C07954=1063.954,157.184,419.924,172.572,29.791,155.478
C07955=1063.959,157.433,419.903,172.574,29.794,155.479
C07956=1063.965,157.682,419.880,172.576,29.796,155.479
C07957=1063.971,157.931,419.858,172.578,29.799,155.480
C07958=1063.977,158.179,419.837,172.579,29.802,155.480
C07959=1063.983,158.464,419.812,172.582,29.805,155.481
C07960=1063.990,158.747,419.787,172.584,29.808,155.481
C07961=1063.996,159.031,419.762,172.586,29.812,155.482
C07962=1064.003,159.314,419.737,172.588,29.815,155.482
C07963=1064.009,159.564,419.716,172.590,29.818,155.483
C07964=1064.015,159.813,419.693,172.591,29.820,155.483
C07965=1064.021,160.062,419.671,172.593,29.823,155.483
C07966=1064.027,160.310,419.650,172.596,29.826,155.484
C07967=1064.032,160.560,419.628,172.597,29.829,155.484
C07968=1064.038,160.809,419.606,172.599,29.831,155.485
C07969=1064.045,161.057,419.584,172.601,29.835,155.485
C07970=1064.049,161.306,419.562,172.603,29.837,155.486
C07971=1064.056,161.555,419.540,172.604,29.840,155.486
C07972=1064.060,161.804,419.518,172.607,29.843,155.486
C07973=1064.066,162.053,419.495,172.609,29.846,155.487
C07974=1064.072,162.302,419.474,172.610,29.849,155.487
C07975=1064.077,162.551,419.452,172.612,29.852,155.488
C07976=1064.083,162.800,419.429,172.614,29.855,155.488
C07977=1064.089,163.049,419.407,172.615,29.857,155.489
C07978=1064.094,163.298,419.385,172.618,29.861,155.489
C07979=1064.100,163.547,419.362,172.620,29.864,155.490
C07980=1064.106,163.796,419.341,172.621,29.867,155.490
C07981=1064.112,164.045,419.318,172.623,29.870,155.491
C07982=1064.116,164.294,419.296,172.625,29.872,155.491
C07983=1064.123,164.543,419.274,172.626,29.875,155.491
C07984=1064.128,164.792,419.251,172.629,29.878,155.492
C07985=1064.133,165.041,419.230,172.631,29.881,155.492
C07986=1064.140,165.289,419.207,172.633,29.884,155.493
C07987=1064.145,165.539,419.185,172.634,29.887,155.493
C07988=1064.151,165.788,419.162,172.636,29.890,155.494
C07989=1064.156,166.036,419.141,172.638,29.893,155.494
C07990=1064.162,166.285,419.118,172.640,29.896,155.495
C07991=1064.167,166.535,419.096,172.642,29.898,155.495
C07992=1064.174,166.783,419.073,172.644,29.902,155.496
C07993=1064.179,167.032,419.051,172.645,29.904,155.496
C07994=1064.184,167.281,419.028,172.647,29.907,155.496
C07995=1064.191,167.530,419.007,172.650,29.910,155.497
C07996=1064.196,167.779,418.984,172.652,29.913,155.497
C07997=1064.201,168.028,418.962,172.653,29.916,155.498
C07998=1064.207,168.277,418.939,172.655,29.919,155.498
C07999=1064.213,168.525,418.917,172.657,29.922,155.499
C08000=1064.219,168.775,418.894,172.659,29.925,155.499
C08001=1064.224,169.024,418.872,172.661,29.928,155.500
C08002=1064.230,169.272,418.850,172.663,29.931,155.500
C08003=1064.236,169.521,418.827,172.664,29.934,155.500
C08004=1064.242,169.770,418.804,172.667,29.937,155.501
C08005=1064.247,170.020,418.782,172.669,29.939,155.501
C08006=1064.253,170.268,418.760,172.670,29.943,155.502
C08007=1064.259,170.500,418.739,172.672,29.945,155.502
C08008=1064.264,170.732,418.718,172.674,29.948,155.503
C08009=1064.269,170.965,418.697,172.676,29.951,155.503
C08010=1064.274,171.197,418.676,172.677,29.953,155.503
C08011=1064.280,171.428,418.655,172.679,29.956,155.504
C08012=1064.285,171.661,418.634,172.681,29.959,155.504
C08013=1064.290,171.893,418.613,172.684,29.962,155.505
C08014=1064.296,172.126,418.592,172.685,29.964,155.505
C08015=1064.301,172.374,418.569,172.687,29.967,155.506
C08016=1064.308,172.622,418.547,172.689,29.970,155.506
C08017=1064.313,172.872,418.524,172.690,29.973,155.506
C08018=1064.319,173.121,418.502,172.693,29.976,155.507
C08019=1064.324,173.370,418.479,172.695,29.978,155.507
C08020=1064.331,173.618,418.456,172.696,29.982,155.508
C08021=1064.336,173.868,418.434,172.698,29.984,155.508
C08022=1064.342,174.117,418.411,172.701,29.987,155.509
C08023=1064.349,174.433,418.382,172.703,29.991,155.509
C08024=1064.356,174.751,418.353,172.705,29.994,155.510
C08025=1064.365,175.068,418.325,172.708,29.998,155.510
C08026=1064.371,175.384,418.296,172.710,30.002,155.511
C08027=1064.377,175.633,418.273,172.712,30.005,155.511
C08028=1064.383,175.882,418.250,172.715,30.008,155.512
C08029=1064.389,176.131,418.228,172.716,30.011,155.512
C08030=1064.395,176.379,418.205,172.718,30.014,155.513
C08031=1064.401,176.628,418.182,172.721,30.017,155.513
C08032=1064.407,176.877,418.159,172.723,30.019,155.514
C08033=1064.412,177.126,418.136,172.724,30.023,155.514
C08034=1064.418,177.375,418.113,172.726,30.025,155.515
C08035=1064.424,177.624,418.091,172.729,30.028,155.515
C08036=1064.430,177.873,418.068,172.730,30.031,155.515
C08037=1064.436,178.122,418.045,172.732,30.034,155.516
C08038=1064.441,178.371,418.022,172.735,30.037,155.516
C08039=1064.447,178.620,418.000,172.737,30.040,155.517
C08040=1064.454,178.868,417.977,172.738,30.043,155.517
C08041=1064.459,179.117,417.954,172.740,30.045,155.518
C08042=1064.465,179.366,417.931,172.743,30.048,155.518
C08043=1064.471,179.616,417.908,172.744,30.051,155.519
C08044=1064.477,179.865,417.885,172.746,30.054,155.519
C08045=1064.483,180.114,417.862,172.749,30.057,155.519
C08046=1064.489,180.362,417.840,172.750,30.060,155.520
C08047=1064.495,180.610,417.816,172.752,30.063,155.520
C08048=1064.501,180.859,417.793,172.755,30.066,155.521
C08049=1064.507,181.108,417.770,172.757,30.069,155.521
C08050=1064.512,181.357,417.747,172.758,30.072,155.522
C08051=1064.518,181.606,417.724,172.761,30.075,155.522
C08052=1064.524,181.855,417.701,172.763,30.078,155.523
C08053=1064.530,182.104,417.678,172.764,30.080,155.523
C08054=1064.537,182.353,417.656,172.767,30.083,155.523
C08055=1064.542,182.602,417.633,172.769,30.086,155.524
C08056=1064.549,182.850,417.609,172.771,30.089,155.524
C08057=1064.554,183.099,417.586,172.773,30.092,155.525
C08058=1064.560,183.348,417.563,172.775,30.095,155.525
C08059=1064.566,183.597,417.540,172.777,30.098,155.526
C08060=1064.571,183.846,417.517,172.779,30.101,155.526
C08061=1064.578,184.095,417.494,172.781,30.103,155.526
C08062=1064.585,184.343,417.471,172.783,30.107,155.527
C08063=1064.590,184.592,417.448,172.786,30.109,155.527
C08064=1064.595,184.842,417.424,172.787,30.113,155.528
C08065=1064.601,185.090,417.401,172.789,30.115,155.528
C08066=1064.607,185.339,417.378,172.792,30.119,155.529
C08067=1064.612,185.588,417.354,172.793,30.121,155.529
C08068=1064.618,185.837,417.331,172.795,30.125,155.530
C08069=1064.624,186.085,417.308,172.798,30.128,155.530
C08070=1064.629,186.334,417.284,172.799,30.131,155.531
C08071=1064.635,186.584,417.261,172.801,30.134,155.531
C08072=1064.641,186.832,417.237,172.804,30.137,155.532
C08073=1064.646,187.081,417.214,172.806,30.140,155.532
C08074=1064.652,187.330,417.191,172.807,30.143,155.533
C08075=1064.658,187.579,417.167,172.810,30.146,155.533
C08076=1064.663,187.828,417.143,172.812,30.149,155.534
C08077=1064.669,188.076,417.120,172.813,30.152,155.534
C08078=1064.674,188.325,417.096,172.816,30.155,155.535
C08079=1064.680,188.574,417.073,172.818,30.158,155.535
C08080=1064.686,188.822,417.050,172.820,30.161,155.536
C08081=1064.691,189.072,417.026,172.822,30.165,155.536
C08082=1064.697,189.321,417.002,172.824,30.167,155.536
C08083=1064.703,189.570,416.979,172.827,30.171,155.537
C08084=1064.708,189.818,416.955,172.828,30.173,155.537
C08085=1064.714,190.067,416.932,172.830,30.177,155.538
C08086=1064.719,190.316,416.908,172.833,30.180,155.538
C08087=1064.726,190.598,416.881,172.835,30.183,155.539
C08088=1064.733,190.882,416.854,172.837,30.187,155.540
C08089=1064.740,191.165,416.827,172.840,30.190,155.540
C08090=1064.746,191.448,416.800,172.842,30.194,155.541
C08091=1064.752,191.696,416.777,172.844,30.197,155.541
C08092=1064.758,191.945,416.753,172.846,30.200,155.542
C08093=1064.763,192.194,416.730,172.849,30.203,155.542
C08094=1064.769,192.443,416.706,172.850,30.206,155.543
C08095=1064.775,192.691,416.681,172.853,30.209,155.543
C08096=1064.780,192.940,416.659,172.855,30.212,155.543
C08097=1064.786,193.189,416.634,172.856,30.215,155.544
C08098=1064.792,193.438,416.610,172.859,30.218,155.544
C08099=1064.798,193.687,416.587,172.861,30.221,155.545
C08100=1064.803,193.935,416.563,172.863,30.225,155.545
C08101=1064.809,194.184,416.539,172.865,30.227,155.546
C08102=1064.815,194.434,416.515,172.868,30.231,155.546
C08103=1064.821,194.682,416.492,172.870,30.234,155.547
C08104=1064.826,194.930,416.468,172.871,30.237,155.547
C08105=1064.832,195.179,416.445,172.874,30.240,155.548
C08106=1064.839,195.428,416.421,172.876,30.243,155.548
C08107=1064.844,195.677,416.396,172.878,30.246,155.549
C08108=1064.850,195.925,416.373,172.880,30.249,155.549
C08109=1064.855,196.175,416.349,172.883,30.252,155.550
C08110=1064.862,196.423,416.325,172.885,30.255,155.550
C08111=1064.867,196.672,416.301,172.886,30.258,155.551
C08112=1064.873,196.921,416.277,172.889,30.261,155.551
C08113=1064.878,197.170,416.253,172.891,30.265,155.552
C08114=1064.884,197.418,416.230,172.893,30.267,155.552
C08115=1064.890,197.668,416.205,172.895,30.271,155.553
C08116=1064.896,197.916,416.181,172.898,30.274,155.553
C08117=1064.902,198.165,416.157,172.900,30.277,155.554
C08118=1064.908,198.414,416.133,172.902,30.280,155.554
C08119=1064.914,198.662,416.109,172.904,30.283,155.555
C08120=1064.919,198.911,416.086,172.907,30.286,155.555
C08121=1064.925,199.160,416.061,172.908,30.289,155.556
C08122=1064.931,199.409,416.038,172.910,30.292,155.556
C08123=1064.937,199.658,416.013,172.913,30.295,155.557
C08124=1064.943,199.906,415.989,172.915,30.299,155.557
C08125=1064.949,200.155,415.965,172.917,30.301,155.557
C08126=1064.955,200.404,415.941,172.919,30.305,155.558
C08127=1064.960,200.652,415.917,172.922,30.308,155.558
C08128=1064.967,200.901,415.893,172.923,30.311,155.559
C08129=1064.972,201.150,415.868,172.926,30.314,155.559
C08130=1064.979,201.399,415.844,172.928,30.317,155.560
C08131=1064.984,201.647,415.820,172.931,30.320,155.560
C08132=1064.991,201.896,415.796,172.932,30.323,155.561
C08133=1064.996,202.145,415.772,172.935,30.326,155.561
C08134=1065.002,202.394,415.748,172.937,30.329,155.562
C08135=1065.008,202.643,415.724,172.939,30.333,155.562
C08136=1065.014,202.891,415.699,172.941,30.336,155.563
C08137=1065.019,203.140,415.675,172.944,30.339,155.563
C08138=1065.025,203.389,415.650,172.946,30.342,155.564
C08139=1065.030,203.638,415.626,172.948,30.345,155.564
C08140=1065.037,203.887,415.602,172.950,30.349,155.565
C08141=1065.042,204.135,415.577,172.953,30.352,155.565
C08142=1065.048,204.384,415.553,172.954,30.355,155.566
C08143=1065.053,204.632,415.528,172.957,30.359,155.566
C08144=1065.059,204.882,415.504,172.959,30.361,155.567
C08145=1065.065,205.130,415.480,172.961,30.365,155.567
C08146=1065.071,205.379,415.455,172.963,30.368,155.568
C08147=1065.077,205.627,415.430,172.966,30.371,155.568
C08148=1065.083,205.877,415.406,172.968,30.374,155.569
C08149=1065.088,206.125,415.382,172.970,30.378,155.570
C08150=1065.093,206.374,415.357,172.972,30.380,155.570
C08151=1065.119,207.420,415.254,173.131,30.459,155.576
C08152=1065.125,207.641,415.232,173.133,30.463,155.576
C08153=1065.129,207.862,415.209,173.135,30.467,155.577
C08154=1065.134,208.083,415.187,173.137,30.470,155.578
C08155=1065.140,208.305,415.164,173.139,30.474,155.578
C08156=1065.146,208.526,415.142,173.141,30.478,155.579
C08157=1065.150,208.746,415.119,173.142,30.481,155.580
C08158=1065.156,208.968,415.097,173.144,30.485,155.580
C08159=1065.162,209.188,415.074,173.146,30.488,155.581
C08160=1065.168,209.437,415.048,173.147,30.493,155.582
C08161=1065.174,209.685,415.023,173.149,30.496,155.582
C08162=1065.179,209.934,414.997,173.152,30.501,155.583
C08163=1065.185,210.182,414.972,173.154,30.504,155.584
C08164=1065.191,210.431,414.947,173.155,30.509,155.584
C08165=1065.197,210.680,414.921,173.158,30.513,155.585
C08166=1065.204,210.928,414.896,173.159,30.517,155.586
C08167=1065.209,211.177,414.870,173.161,30.521,155.586
C08168=1065.215,211.426,414.845,173.164,30.525,155.587
C08169=1065.222,211.675,414.819,173.165,30.529,155.588
C08170=1065.227,211.924,414.793,173.167,30.533,155.589
C08171=1065.233,212.172,414.768,173.169,30.537,155.589
C08172=1065.239,212.421,414.743,173.171,30.542,155.590
C08173=1065.246,212.670,414.717,173.173,30.545,155.591
C08174=1065.251,212.918,414.691,173.175,30.550,155.592
C08175=1065.257,213.166,414.666,173.178,30.553,155.592
C08176=1065.263,213.415,414.640,173.179,30.558,155.593
C08177=1065.269,213.664,414.615,173.181,30.562,155.594
C08178=1065.275,213.912,414.589,173.183,30.566,155.594
C08179=1065.281,214.161,414.563,173.185,30.570,155.595
C08180=1065.287,214.409,414.537,173.187,30.574,155.596
C08181=1065.292,214.658,414.511,173.190,30.578,155.597
C08182=1065.299,214.907,414.486,173.191,30.582,155.597
C08183=1065.305,215.155,414.460,173.193,30.586,155.598
C08184=1065.311,215.404,414.434,173.196,30.590,155.599
C08185=1065.317,215.653,414.409,173.197,30.594,155.599
C08186=1065.322,215.902,414.383,173.200,30.599,155.600
C08187=1065.329,216.150,414.357,173.202,30.602,155.601
C08188=1065.334,216.399,414.331,173.203,30.607,155.602
C08189=1065.340,216.647,414.305,173.206,30.611,155.602
C08190=1065.347,216.895,414.279,173.208,30.615,155.603
C08191=1065.352,217.144,414.253,173.209,30.619,155.604
C08192=1065.359,217.393,414.228,173.212,30.623,155.604
C08193=1065.364,217.641,414.201,173.214,30.627,155.605
C08194=1065.371,217.890,414.176,173.215,30.631,155.606
C08195=1065.376,218.138,414.149,173.218,30.635,155.607
C08196=1065.383,218.387,414.124,173.220,30.639,155.607
C08197=1065.388,218.636,414.098,173.222,30.643,155.608
C08198=1065.395,218.884,414.072,173.224,30.647,155.609
C08199=1065.400,219.133,414.046,173.226,30.651,155.609
C08200=1065.406,219.381,414.020,173.228,30.655,155.610
C08201=1065.412,219.630,413.994,173.230,30.659,155.611
C08202=1065.418,219.878,413.968,173.232,30.663,155.612
C08203=1065.425,220.128,413.942,173.234,30.667,155.612
C08204=1065.431,220.376,413.916,173.236,30.671,155.613
C08205=1065.437,220.625,413.890,173.239,30.675,155.614
C08206=1065.443,220.873,413.864,173.241,30.679,155.614
C08207=1065.449,221.122,413.838,173.242,30.683,155.615
C08208=1065.455,221.345,413.814,173.245,30.687,155.616
C08209=1065.460,221.569,413.790,173.247,30.690,155.616
C08210=1065.465,221.792,413.768,173.248,30.694,155.617
C08211=1065.470,222.015,413.743,173.250,30.698,155.618
C08212=1065.475,222.239,413.720,173.252,30.702,155.618
C08213=1065.481,222.462,413.697,173.254,30.705,155.619
C08214=1065.486,222.685,413.672,173.255,30.708,155.619
C08215=1065.492,222.909,413.649,173.258,30.712,155.620
C08216=1065.498,223.157,413.623,173.260,30.717,155.621
C08217=1065.503,223.406,413.597,173.261,30.720,155.622
C08218=1065.509,223.655,413.570,173.264,30.724,155.622
C08219=1065.516,223.903,413.544,173.266,30.729,155.623
C08220=1065.521,224.152,413.518,173.268,30.732,155.624
C08221=1065.527,224.400,413.492,173.270,30.737,155.624
C08222=1065.533,224.649,413.465,173.272,30.740,155.625
C08223=1065.540,224.897,413.438,173.275,30.745,155.626
C08224=1065.545,225.146,413.413,173.276,30.749,155.627
C08225=1065.551,225.394,413.386,173.279,30.753,155.627
C08226=1065.557,225.643,413.359,173.281,30.757,155.628
C08227=1065.563,225.891,413.333,173.283,30.761,155.629
C08228=1065.569,226.140,413.307,173.285,30.765,155.629
C08229=1065.575,226.389,413.280,173.287,30.769,155.630
C08230=1065.581,226.637,413.254,173.289,30.773,155.631
C08231=1065.587,226.885,413.228,173.291,30.777,155.632
C08232=1065.593,227.134,413.201,173.294,30.781,155.632
C08233=1065.600,227.383,413.174,173.296,30.784,155.633
C08234=1065.605,227.632,413.148,173.298,30.789,155.634
C08235=1065.611,227.880,413.121,173.300,30.793,155.634
C08236=1065.617,228.128,413.095,173.303,30.797,155.635
C08237=1065.624,228.377,413.068,173.304,30.801,155.636
C08238=1065.629,228.625,413.042,173.306,30.805,155.636
C08239=1065.635,228.874,413.015,173.309,30.808,155.637
C08240=1065.641,229.122,412.988,173.311,30.813,155.638
C08241=1065.648,229.371,412.962,173.313,30.817,155.638
C08242=1065.654,229.619,412.935,173.315,30.820,155.639
C08243=1065.660,229.868,412.909,173.318,30.825,155.640
C08244=1065.665,230.116,412.882,173.319,30.828,155.641
C08245=1065.672,230.365,412.855,173.322,30.833,155.641
C08246=1065.678,230.613,412.828,173.324,30.837,155.642
C08247=1065.683,230.862,412.802,173.327,30.840,155.643
C08248=1065.689,231.110,412.775,173.328,30.845,155.643
C08249=1065.696,231.359,412.748,173.331,30.849,155.644
C08250=1065.701,231.608,412.721,173.333,30.853,155.645
C08251=1065.707,231.856,412.695,173.335,30.857,155.646
C08252=1065.713,232.105,412.668,173.337,30.860,155.646
C08253=1065.719,232.353,412.641,173.339,30.865,155.647
C08254=1065.725,232.602,412.614,173.341,30.869,155.648
C08255=1065.732,232.850,412.587,173.343,30.872,155.648
C08256=1065.737,233.098,412.560,173.346,30.877,155.649
C08257=1065.743,233.347,412.533,173.348,30.881,155.650
C08258=1065.749,233.595,412.507,173.350,30.884,155.650
C08259=1065.755,233.844,412.480,173.352,30.889,155.651
C08260=1065.760,234.093,412.452,173.355,30.893,155.652
C08261=1065.767,234.341,412.425,173.357,30.897,155.653
C08262=1065.773,234.590,412.398,173.359,30.901,155.653
C08263=1065.779,234.838,412.371,173.361,30.904,155.654
C08264=1065.787,235.172,412.335,173.365,30.910,155.655
C08265=1065.795,235.505,412.299,173.367,30.916,155.656
C08266=1065.803,235.839,412.263,173.370,30.921,155.657
C08267=1065.811,236.172,412.226,173.373,30.926,155.658
C08268=1065.817,236.421,412.199,173.375,30.930,155.658
C08269=1065.823,236.669,412.172,173.378,30.934,155.659
C08270=1065.829,236.918,412.144,173.380,30.938,155.660
C08271=1065.835,237.167,412.117,173.382,30.942,155.661
C08272=1065.840,237.415,412.091,173.384,30.946,155.661
C08273=1065.847,237.663,412.063,173.387,30.950,155.662
C08274=1065.853,237.912,412.036,173.390,30.954,155.663
C08275=1065.859,238.161,412.009,173.391,30.958,155.663
C08276=1065.867,238.514,411.970,173.395,30.963,155.664
C08277=1065.876,238.868,411.931,173.397,30.969,155.665
C08278=1065.884,239.221,411.892,173.401,30.975,155.666
C08279=1065.893,239.575,411.853,173.404,30.980,155.667
C08280=1065.899,239.823,411.826,173.406,30.985,155.668
C08281=1065.905,240.072,411.798,173.409,30.989,155.669
C08282=1065.911,240.320,411.771,173.411,30.992,155.669
C08283=1065.917,240.568,411.744,173.414,30.997,155.670
C08284=1065.923,240.817,411.717,173.415,31.000,155.671
C08285=1065.929,241.065,411.689,173.418,31.004,155.672
C08286=1065.935,241.314,411.662,173.420,31.009,155.672
C08287=1065.941,241.562,411.635,173.423,31.012,155.673
C08288=1065.948,241.811,411.608,173.424,31.016,155.674
C08289=1065.953,242.059,411.580,173.427,31.020,155.674
C08290=1065.960,242.307,411.552,173.430,31.024,155.675
C08291=1065.966,242.556,411.525,173.432,31.028,155.676
C08292=1065.971,242.804,411.497,173.434,31.032,155.677
C08293=1065.977,243.052,411.470,173.436,31.036,155.677
C08294=1065.983,243.302,411.442,173.439,31.040,155.678
C08295=1065.989,243.549,411.415,173.440,31.044,155.679
C08296=1065.995,243.798,411.386,173.443,31.048,155.679
C08297=1066.001,244.046,411.360,173.446,31.052,155.680
C08298=1066.007,244.295,411.331,173.448,31.056,155.681
C08299=1066.013,244.543,411.304,173.450,31.060,155.681
C08300=1066.019,244.792,411.276,173.452,31.064,155.682
C08301=1066.025,245.041,411.249,173.455,31.068,155.683
C08302=1066.030,245.289,411.221,173.458,31.072,155.684
C08303=1066.037,245.537,411.193,173.459,31.076,155.684
C08304=1066.042,245.785,411.165,173.462,31.080,155.685
C08305=1066.049,246.034,411.137,173.464,31.084,155.686
C08306=1066.055,246.282,411.109,173.467,31.088,155.686
C08307=1066.061,246.531,411.082,173.468,31.092,155.687
C08308=1066.066,246.779,411.054,173.471,31.096,155.688
C08309=1066.072,247.028,411.026,173.474,31.100,155.689
C08310=1066.078,247.275,410.999,173.476,31.104,155.689
C08311=1066.084,247.524,410.970,173.478,31.108,155.690
C08312=1066.090,247.773,410.942,173.480,31.112,155.691
C08313=1066.096,248.021,410.915,173.483,31.116,155.691
C08314=1066.102,248.269,410.886,173.486,31.120,155.692
C08315=1066.107,248.517,410.858,173.487,31.124,155.693
C08316=1066.113,248.734,410.834,173.490,31.128,155.693
C08317=1066.118,248.950,410.810,173.492,31.131,155.694
C08318=1066.123,249.166,410.785,173.494,31.135,155.695
C08319=1066.128,249.383,410.761,173.495,31.138,155.695
C08320=1066.133,249.599,410.736,173.498,31.141,155.696
C08321=1066.138,249.815,410.712,173.500,31.145,155.697
C08322=1066.144,250.032,410.688,173.502,31.149,155.697
C08323=1066.148,250.247,410.663,173.505,31.152,155.698
C08324=1066.154,250.496,410.635,173.506,31.156,155.699
C08325=1066.161,250.744,410.607,173.509,31.160,155.699
C08326=1066.166,250.992,410.579,173.511,31.164,155.700
C08327=1066.172,251.241,410.551,173.514,31.168,155.701
C08328=1066.178,251.490,410.523,173.516,31.172,155.701
C08329=1066.184,251.737,410.495,173.518,31.176,155.702
C08330=1066.191,251.985,410.466,173.521,31.180,155.703
C08331=1066.196,252.234,410.438,173.524,31.184,155.703
C08332=1066.202,252.482,410.410,173.525,31.188,155.704
C08333=1066.208,252.731,410.382,173.528,31.192,155.705
C08334=1066.214,252.979,410.354,173.531,31.196,155.706
C08335=1066.220,253.227,410.325,173.533,31.200,155.706
C08336=1066.226,253.476,410.297,173.535,31.204,155.707
C08337=1066.232,253.724,410.269,173.538,31.208,155.708
C08338=1066.237,253.972,410.241,173.540,31.212,155.708
C08339=1066.244,254.220,410.212,173.543,31.216,155.709
C08340=1066.250,254.469,410.184,173.545,31.220,155.710
C08341=1066.256,254.718,410.155,173.547,31.224,155.711
C08342=1066.262,254.966,410.127,173.550,31.228,155.711
C08343=1066.268,255.214,410.098,173.553,31.232,155.712
C08344=1066.274,255.463,410.070,173.554,31.236,155.713
C08345=1066.280,255.711,410.042,173.557,31.240,155.713
C08346=1066.286,255.959,410.014,173.560,31.244,155.714
C08347=1066.292,256.207,409.985,173.562,31.248,155.715
C08348=1066.298,256.455,409.956,173.564,31.252,155.715
C08349=1066.304,256.704,409.928,173.567,31.255,155.716
C08350=1066.310,256.953,409.900,173.569,31.260,155.717
C08351=1066.317,257.200,409.872,173.572,31.263,155.718
C08352=1066.322,257.449,409.843,173.575,31.267,155.718
C08353=1066.329,257.697,409.814,173.576,31.272,155.719
C08354=1066.335,257.946,409.786,173.579,31.275,155.720
C08355=1066.341,258.194,409.757,173.582,31.279,155.720
C08356=1066.347,258.443,409.729,173.585,31.284,155.721
C08357=1066.352,258.690,409.700,173.586,31.287,155.722
C08358=1066.359,258.938,409.672,173.589,31.291,155.722
C08359=1066.365,259.187,409.643,173.592,31.295,155.723
C08360=1066.371,259.435,409.615,173.594,31.299,155.724
C08361=1066.378,259.683,409.586,173.596,31.303,155.725
C08362=1066.384,259.932,409.557,173.599,31.307,155.725
C08363=1066.390,260.180,409.528,173.602,31.311,155.726
C08364=1066.396,260.429,409.500,173.604,31.315,155.727
C08365=1066.401,260.677,409.471,173.607,31.319,155.727
C08366=1066.408,260.925,409.442,173.609,31.322,155.728
C08367=1066.414,261.173,409.415,173.612,31.327,155.729
C08368=1066.421,261.421,409.386,173.614,31.330,155.729
C08369=1066.427,261.669,409.357,173.617,31.334,155.730
C08370=1066.433,261.918,409.328,173.619,31.338,155.731
C08371=1066.439,262.166,409.299,173.622,31.342,155.732
C08372=1066.445,262.382,409.274,173.624,31.346,155.732
C08373=1066.449,262.597,409.249,173.626,31.349,155.733
C08374=1066.455,262.811,409.224,173.629,31.352,155.733
C08375=1066.461,263.027,409.200,173.630,31.356,155.734
C08376=1066.466,263.241,409.174,173.633,31.359,155.735
C08377=1066.471,263.457,409.149,173.635,31.362,155.735
C08378=1066.476,263.672,409.124,173.637,31.366,155.736
C08379=1066.482,263.888,409.099,173.640,31.369,155.736
C08380=1066.487,264.135,409.071,173.641,31.374,155.737
C08381=1066.493,264.383,409.042,173.644,31.377,155.738
C08382=1066.500,264.631,409.012,173.647,31.381,155.738
C08383=1066.505,264.880,408.983,173.650,31.386,155.739
C08384=1066.511,265.128,408.954,173.652,31.389,155.740
C08385=1066.518,265.376,408.925,173.654,31.394,155.741
C08386=1066.524,265.624,408.896,173.657,31.397,155.741
C08387=1066.529,265.873,408.867,173.660,31.401,155.742
C08388=1066.535,266.121,408.838,173.663,31.406,155.743
C08389=1066.542,266.369,408.809,173.665,31.409,155.744
C08390=1066.548,266.618,408.780,173.667,31.414,155.744
C08391=1066.553,266.866,408.750,173.670,31.417,155.745
C08392=1066.560,267.114,408.721,173.673,31.421,155.746
C08393=1066.566,267.362,408.692,173.675,31.425,155.746
C08394=1066.572,267.610,408.663,173.677,31.429,155.747
C08395=1066.578,267.859,408.633,173.680,31.434,155.748
C08396=1066.584,268.107,408.604,173.683,31.437,155.749
C08397=1066.590,268.355,408.575,173.686,31.441,155.749
C08398=1066.596,268.604,408.546,173.688,31.445,155.750
C08399=1066.602,268.851,408.516,173.690,31.449,155.751
C08400=1066.609,269.099,408.487,173.693,31.454,155.751
C08401=1066.614,269.348,408.457,173.696,31.457,155.752
C08402=1066.620,269.596,408.428,173.699,31.461,155.753
C08403=1066.627,269.844,408.399,173.701,31.465,155.754
C08404=1066.632,270.092,408.369,173.703,31.469,155.754
C08405=1066.638,270.341,408.340,173.706,31.474,155.755
C08406=1066.644,270.588,408.310,173.709,31.477,155.756
C08407=1066.650,270.836,408.281,173.712,31.482,155.756
C08408=1066.657,271.085,408.252,173.714,31.485,155.757
C08409=1066.663,271.334,408.222,173.716,31.489,155.758
C08410=1066.669,271.582,408.193,173.719,31.493,155.759
C08411=1066.675,271.830,408.163,173.722,31.497,155.759
C08412=1066.681,272.078,408.134,173.725,31.502,155.760
C08413=1066.687,272.326,408.104,173.727,31.505,155.761
C08414=1066.693,272.574,408.074,173.729,31.510,155.762
C08415=1066.699,272.822,408.044,173.732,31.513,155.762
C08416=1066.705,273.070,408.015,173.735,31.517,155.763
C08417=1066.711,273.318,407.985,173.738,31.522,155.764
C08418=1066.717,273.566,407.956,173.740,31.525,155.764
C08419=1066.723,273.815,407.926,173.743,31.530,155.765
C08420=1066.730,274.063,407.896,173.746,31.533,155.766
C08421=1066.735,274.311,407.867,173.748,31.538,155.767
C08422=1066.742,274.559,407.837,173.751,31.541,155.767
C08423=1066.747,274.807,407.807,173.753,31.546,155.768
C08424=1066.753,275.056,407.778,173.756,31.550,155.769
C08425=1066.759,275.303,407.748,173.759,31.554,155.769
C08426=1066.765,275.552,407.718,173.762,31.558,155.770
C08427=1066.772,275.800,407.688,173.765,31.562,155.771
C08428=1066.776,276.017,407.662,173.766,31.566,155.772
C08429=1066.782,276.234,407.636,173.769,31.569,155.772
C08430=1066.787,276.450,407.609,173.771,31.573,155.773
C08431=1066.792,276.667,407.583,173.774,31.576,155.774
C08432=1066.798,276.884,407.558,173.776,31.579,155.774
C08433=1066.803,277.101,407.532,173.779,31.583,155.775
C08434=1066.808,277.317,407.505,173.780,31.587,155.775
C08435=1066.814,277.534,407.479,173.783,31.590,155.776
C08436=1066.820,277.783,407.449,173.785,31.594,155.777
C08437=1066.826,278.031,407.419,173.788,31.598,155.777
C08438=1066.832,278.279,407.389,173.791,31.602,155.778
C08439=1066.838,278.527,407.360,173.793,31.606,155.779
C08440=1066.843,278.775,407.329,173.796,31.610,155.780
C08441=1066.851,279.023,407.299,173.799,31.614,155.780
C08442=1066.856,279.271,407.269,173.802,31.619,155.781
C08443=1066.862,279.520,407.239,173.805,31.622,155.782
C08444=1066.868,279.767,407.209,173.807,31.627,155.783
C08445=1066.875,280.016,407.179,173.810,31.630,155.783
C08446=1066.880,280.264,407.149,173.812,31.635,155.784
C08447=1066.886,280.512,407.119,173.815,31.638,155.785
C08448=1066.893,280.760,407.088,173.818,31.643,155.786
C08449=1066.898,281.008,407.058,173.821,31.647,155.786
C08450=1066.904,281.256,407.027,173.823,31.651,155.787
C08451=1066.911,281.504,406.998,173.826,31.655,155.788
C08452=1066.917,281.753,406.967,173.829,31.659,155.789
C08453=1066.923,282.000,406.937,173.832,31.663,155.789
C08454=1066.929,282.248,406.907,173.835,31.668,155.790
C08455=1066.934,282.496,406.876,173.837,31.671,155.791
C08456=1066.941,282.745,406.846,173.840,31.676,155.791
C08457=1066.947,282.992,406.815,173.842,31.680,155.792
C08458=1066.952,283.240,406.785,173.845,31.684,155.793
C08459=1066.959,283.489,406.754,173.848,31.688,155.794
C08460=1066.965,283.737,406.724,173.851,31.692,155.795
C08461=1066.971,283.984,406.694,173.853,31.696,155.795
C08462=1066.977,284.233,406.663,173.856,31.700,155.796
C08463=1066.983,284.481,406.632,173.859,31.704,155.797
C08464=1066.989,284.729,406.602,173.862,31.708,155.797
C08465=1066.995,284.977,406.571,173.865,31.713,155.798
C08466=1067.001,285.225,406.541,173.867,31.716,155.799
C08467=1067.008,285.473,406.511,173.870,31.721,155.800
C08468=1067.014,285.721,406.481,173.873,31.725,155.800
C08469=1067.020,285.969,406.450,173.876,31.729,155.801
C08470=1067.026,286.217,406.420,173.879,31.733,155.802
C08471=1067.032,286.465,406.389,173.882,31.737,155.803
C08472=1067.039,286.713,406.358,173.884,31.741,155.803
C08473=1067.044,286.961,406.327,173.887,31.745,155.804
C08474=1067.050,287.209,406.297,173.890,31.749,155.805
C08475=1067.057,287.457,406.266,173.893,31.754,155.806
C08476=1067.062,287.705,406.236,173.896,31.757,155.806
C08477=1067.069,287.954,406.205,173.898,31.762,155.807
C08478=1067.075,288.201,406.174,173.901,31.766,155.808
C08479=1067.081,288.449,406.143,173.904,31.770,155.809
C08480=1067.087,288.697,406.113,173.907,31.774,155.809
C08481=1067.093,288.945,406.081,173.910,31.778,155.810
C08482=1067.099,289.193,406.051,173.913,31.782,155.811
C08483=1067.105,289.442,406.020,173.915,31.786,155.812
C08484=1067.111,289.663,405.993,173.917,31.790,155.812
C08485=1067.116,289.885,405.965,173.920,31.794,155.813
C08486=1067.122,290.107,405.937,173.923,31.798,155.814
C08487=1067.127,290.329,405.909,173.925,31.801,155.814
C08488=1067.132,290.552,405.881,173.928,31.805,155.815
C08489=1067.138,290.773,405.854,173.931,31.809,155.816
C08490=1067.143,290.996,405.826,173.932,31.812,155.816
C08491=1067.149,291.218,405.799,173.935,31.816,155.817
C08492=1067.156,291.465,405.768,173.938,31.820,155.818
C08493=1067.161,291.714,405.737,173.941,31.825,155.819
C08494=1067.167,291.962,405.705,173.944,31.828,155.819
C08495=1067.173,292.209,405.675,173.947,31.833,155.820
C08496=1067.180,292.457,405.644,173.949,31.837,155.821
C08497=1067.185,292.705,405.613,173.952,31.841,155.822
C08498=1067.192,292.953,405.581,173.955,31.845,155.822
C08499=1067.198,293.201,405.551,173.958,31.849,155.823
C08500=1067.204,293.449,405.519,173.961,31.854,155.824
C08501=1067.210,293.696,405.488,173.964,31.858,155.825
C08502=1067.216,293.945,405.457,173.966,31.862,155.826
C08503=1067.223,294.193,405.426,173.970,31.866,155.826
C08504=1067.228,294.441,405.395,173.973,31.870,155.827
C08505=1067.235,294.689,405.363,173.976,31.875,155.828
C08506=1067.241,294.936,405.332,173.979,31.879,155.829
C08507=1067.246,295.185,405.301,173.982,31.883,155.829
C08508=1067.253,295.433,405.269,173.984,31.887,155.830
C08509=1067.259,295.680,405.238,173.987,31.891,155.831
C08510=1067.265,295.929,405.207,173.990,31.896,155.832
C08511=1067.271,296.176,405.176,173.993,31.900,155.833
C08512=1067.277,296.424,405.144,173.996,31.904,155.833
C08513=1067.284,296.672,405.113,173.999,31.908,155.834
C08514=1067.289,296.920,405.081,174.001,31.912,155.835
C08515=1067.296,297.168,405.050,174.004,31.917,155.836
C08516=1067.301,297.416,405.018,174.007,31.921,155.836
C08517=1067.308,297.664,404.987,174.010,31.925,155.837
C08518=1067.314,297.912,404.955,174.014,31.930,155.838
C08519=1067.319,298.159,404.923,174.017,31.934,155.839
C08520=1067.326,298.407,404.892,174.020,31.938,155.840
C08521=1067.331,298.655,404.860,174.022,31.942,155.840
C08522=1067.337,298.903,404.828,174.025,31.947,155.841
C08523=1067.344,299.151,404.797,174.028,31.951,155.842
C08524=1067.349,299.398,404.765,174.031,31.955,155.843
C08525=1067.355,299.647,404.733,174.034,31.959,155.844
C08526=1067.362,299.895,404.702,174.037,31.964,155.844
C08527=1067.367,300.142,404.670,174.039,31.968,155.845
C08528=1067.373,300.390,404.638,174.042,31.972,155.846
C08529=1067.379,300.637,404.607,174.046,31.977,155.847
C08530=1067.385,300.886,404.575,174.049,31.981,155.848
C08531=1067.391,301.134,404.543,174.052,31.985,155.848
C08532=1067.397,301.382,404.511,174.055,31.990,155.849
C08533=1067.404,301.629,404.480,174.058,31.994,155.850
C08534=1067.410,301.878,404.448,174.060,31.999,155.851
C08535=1067.416,302.126,404.416,174.063,32.003,155.852
C08536=1067.421,302.373,404.384,174.066,32.007,155.852
C08537=1067.428,302.621,404.352,174.069,32.011,155.853
C08538=1067.434,302.869,404.320,174.073,32.016,155.854
C08539=1067.440,303.117,404.288,174.076,32.020,155.855
C08540=1067.445,303.346,404.258,174.079,32.024,155.856
C08541=1067.451,303.576,404.228,174.081,32.028,155.856
C08542=1067.457,303.805,404.200,174.083,32.032,155.857
C08543=1067.463,304.034,404.170,174.086,32.036,155.858
C08544=1067.469,304.264,404.140,174.089,32.040,155.859
C08545=1067.474,304.493,404.110,174.092,32.044,155.859
C08546=1067.479,304.724,404.081,174.095,32.048,155.860
C08547=1067.485,304.953,404.051,174.098,32.052,155.861
C08548=1067.491,305.200,404.019,174.101,32.056,155.862
C08549=1067.497,305.448,403.987,174.103,32.060,155.862
C08550=1067.504,305.696,403.955,174.107,32.065,155.863
C08551=1067.510,305.944,403.923,174.110,32.070,155.864
C08552=1067.516,306.192,403.891,174.113,32.074,155.865
C08553=1067.522,306.440,403.858,174.116,32.078,155.866
C08554=1067.528,306.687,403.826,174.119,32.082,155.867
C08555=1067.535,306.935,403.794,174.123,32.087,155.867
C08556=1067.541,307.183,403.762,174.125,32.091,155.868
C08557=1067.547,307.431,403.730,174.128,32.095,155.869
C08558=1067.553,307.679,403.697,174.131,32.100,155.870
C08559=1067.559,307.927,403.665,174.134,32.104,155.871
C08560=1067.565,308.174,403.632,174.138,32.109,155.871
C08561=1067.572,308.422,403.601,174.141,32.113,155.872
C08562=1067.578,308.670,403.568,174.144,32.117,155.873
C08563=1067.585,308.917,403.536,174.147,32.122,155.874
C08564=1067.591,309.166,403.504,174.149,32.126,155.875
C08565=1067.597,309.413,403.471,174.153,32.130,155.875
C08566=1067.603,309.661,403.439,174.156,32.135,155.876
C08567=1067.609,309.909,403.406,174.159,32.139,155.877
C08568=1067.616,310.156,403.374,174.162,32.144,155.878
C08569=1067.622,310.405,403.342,174.166,32.148,155.879
C08570=1067.628,310.652,403.309,174.169,32.152,155.880
C08571=1067.635,310.900,403.276,174.172,32.156,155.880
C08572=1067.641,311.148,403.244,174.174,32.161,155.881
C08573=1067.647,311.396,403.212,174.177,32.166,155.882
C08574=1067.653,311.643,403.179,174.181,32.170,155.883
C08575=1067.659,311.891,403.147,174.184,32.174,155.884
C08576=1067.666,312.139,403.114,174.187,32.178,155.885
C08577=1067.673,312.386,403.082,174.190,32.183,155.885
C08578=1067.679,312.634,403.049,174.194,32.187,155.886
C08579=1067.685,312.881,403.016,174.197,32.192,155.887
C08580=1067.691,313.130,402.984,174.199,32.196,155.888
C08581=1067.697,313.377,402.952,174.203,32.200,155.889
C08582=1067.704,313.626,402.919,174.206,32.205,155.889
C08583=1067.711,313.873,402.886,174.209,32.209,155.890
C08584=1067.717,314.121,402.853,174.212,32.214,155.891
C08585=1067.723,314.368,402.820,174.216,32.218,155.892
C08586=1067.729,314.616,402.787,174.219,32.223,155.893
C08587=1067.735,314.864,402.754,174.222,32.227,155.894
C08588=1067.741,315.111,402.722,174.224,32.232,155.895
C08589=1067.747,315.359,402.688,174.228,32.236,155.895
C08590=1067.753,315.607,402.655,174.231,32.241,155.896
C08591=1067.759,315.855,402.622,174.234,32.245,155.897
C08592=1067.765,316.102,402.589,174.237,32.250,155.898
C08593=1067.771,316.350,402.557,174.241,32.254,155.899
C08594=1067.777,316.598,402.523,174.244,32.259,155.900
C08595=1067.783,316.845,402.491,174.247,32.264,155.901
C08596=1067.790,317.077,402.459,174.250,32.268,155.902
C08597=1067.795,317.308,402.428,174.252,32.272,155.902
C08598=1067.801,317.540,402.397,174.255,32.277,155.903
C08599=1067.806,317.771,402.367,174.258,32.281,155.904
C08600=1067.812,318.002,402.336,174.262,32.285,155.905
C08601=1067.818,318.234,402.304,174.265,32.289,155.906
C08602=1067.823,318.464,402.273,174.268,32.294,155.906
C08603=1067.829,318.697,402.243,174.271,32.298,155.907
C08604=1067.835,318.944,402.209,174.274,32.303,155.908
C08605=1067.841,319.191,402.176,174.277,32.307,155.909
C08606=1067.848,319.439,402.143,174.281,32.312,155.910
C08607=1067.853,319.687,402.110,174.283,32.317,155.911
C08608=1067.860,319.935,402.076,174.286,32.321,155.912
C08609=1067.866,320.183,402.043,174.290,32.326,155.913
C08610=1067.872,320.430,402.010,174.293,32.331,155.913
C08611=1067.878,320.677,401.976,174.296,32.335,155.914
C08612=1067.884,320.925,401.943,174.300,32.340,155.915
C08613=1067.891,321.173,401.909,174.303,32.344,155.916
C08614=1067.897,321.421,401.876,174.306,32.349,155.917
C08615=1067.903,321.668,401.842,174.310,32.354,155.918
C08616=1067.910,321.916,401.809,174.313,32.358,155.919
C08617=1067.915,322.164,401.775,174.316,32.363,155.920
C08618=1067.922,322.411,401.742,174.319,32.367,155.921
C08619=1067.928,322.659,401.709,174.322,32.372,155.921
C08620=1067.935,322.907,401.675,174.325,32.377,155.922
C08621=1067.940,323.154,401.641,174.329,32.381,155.923
C08622=1067.947,323.401,401.608,174.332,32.386,155.924
C08623=1067.953,323.650,401.574,174.336,32.391,155.925
C08624=1067.960,323.897,401.541,174.339,32.395,155.926
C08625=1067.966,324.146,401.507,174.342,32.400,155.927
C08626=1067.972,324.393,401.473,174.346,32.405,155.928
C08627=1067.978,324.640,401.440,174.349,32.410,155.929
C08628=1067.985,324.889,401.406,174.351,32.414,155.930
C08629=1067.991,325.135,401.372,174.355,32.419,155.930
C08630=1067.998,325.383,401.338,174.358,32.423,155.931
C08631=1068.004,325.631,401.305,174.362,32.428,155.932
C08632=1068.010,325.878,401.271,174.365,32.433,155.933
C08633=1068.016,326.126,401.237,174.368,32.437,155.934
C08634=1068.022,326.374,401.204,174.372,32.442,155.935
C08635=1068.029,326.622,401.170,174.375,32.447,155.936
C08636=1068.036,326.869,401.136,174.379,32.452,155.937
C08637=1068.042,327.117,401.102,174.382,32.456,155.938
C08638=1068.049,327.364,401.068,174.386,32.461,155.939
C08639=1068.055,327.612,401.035,174.389,32.466,155.939
C08640=1068.061,327.860,401.000,174.392,32.470,155.940
C08641=1068.068,328.107,400.967,174.395,32.475,155.941
C08642=1068.074,328.355,400.933,174.398,32.480,155.942
C08643=1068.080,328.603,400.898,174.402,32.485,155.943
C08644=1068.087,328.850,400.865,174.405,32.489,155.944
C08645=1068.093,329.098,400.830,174.409,32.494,155.945
C08646=1068.100,329.346,400.797,174.412,32.499,155.946
C08647=1068.106,329.593,400.763,174.416,32.503,155.947
C08648=1068.112,329.841,400.729,174.419,32.508,155.948
C08649=1068.119,330.088,400.695,174.422,32.513,155.949
C08650=1068.125,330.336,400.661,174.426,32.518,155.950
C08651=1068.132,330.584,400.626,174.429,32.523,155.951
C08652=1068.138,330.812,400.595,174.433,32.527,155.951
C08653=1068.145,331.040,400.563,174.436,32.532,155.952
C08654=1068.150,331.268,400.532,174.438,32.536,155.953
C08655=1068.155,331.497,400.500,174.441,32.540,155.954
C08656=1068.161,331.725,400.469,174.444,32.545,155.955
C08657=1068.167,331.953,400.437,174.448,32.550,155.956
C08658=1068.172,332.181,400.405,174.451,32.554,155.957
C08659=1068.179,332.409,400.374,174.454,32.558,155.958
C08660=1068.185,332.657,400.339,174.458,32.563,155.958
C08661=1068.191,332.905,400.305,174.461,32.569,155.959
C08662=1068.198,333.153,400.271,174.464,32.573,155.960
C08663=1068.204,333.399,400.236,174.468,32.578,155.961
C08664=1068.210,333.647,400.201,174.471,32.583,155.962
C08665=1068.217,333.895,400.167,174.475,32.588,155.963
C08666=1068.223,334.142,400.132,174.478,32.593,155.964
C08667=1068.229,334.390,400.098,174.482,32.598,155.965
C08668=1068.236,334.638,400.063,174.486,32.603,155.966
C08669=1068.242,334.885,400.029,174.489,32.608,155.967
C08670=1068.249,335.133,399.994,174.493,32.613,155.968
C08671=1068.255,335.381,399.960,174.495,32.618,155.969
C08672=1068.261,335.627,399.925,174.499,32.623,155.970
C08673=1068.267,335.876,399.890,174.502,32.628,155.971
C08674=1068.274,336.123,399.855,174.506,32.632,155.972
C08675=1068.279,336.370,399.821,174.509,32.638,155.973
C08676=1068.286,336.618,399.786,174.513,32.643,155.974
C08677=1068.293,336.866,399.751,174.516,32.647,155.975
C08678=1068.299,337.113,399.716,174.520,32.653,155.976
C08679=1068.305,337.360,399.682,174.523,32.657,155.977
C08680=1068.312,337.608,399.647,174.527,32.663,155.978
C08681=1068.319,337.856,399.613,174.531,32.668,155.979
C08682=1068.325,338.103,399.577,174.534,32.673,155.980
C08683=1068.331,338.350,399.542,174.538,32.678,155.981
C08684=1068.337,338.598,399.508,174.541,32.683,155.982
C08685=1068.344,338.845,399.473,174.545,32.688,155.983
C08686=1068.350,339.093,399.437,174.548,32.693,155.984
C08687=1068.356,339.340,399.403,174.552,32.698,155.985
C08688=1068.363,339.588,399.368,174.555,32.703,155.986
C08689=1068.369,339.835,399.332,174.559,32.708,155.987
C08690=1068.375,340.083,399.297,174.563,32.713,155.988
C08691=1068.382,340.331,399.262,174.566,32.719,155.989
C08692=1068.389,340.578,399.227,174.570,32.724,155.990
C08693=1068.394,340.825,399.192,174.573,32.729,155.991
C08694=1068.401,341.072,399.157,174.576,32.734,155.992
C08695=1068.408,341.320,399.122,174.580,32.739,155.993
C08696=1068.414,341.567,399.086,174.583,32.744,155.994
C08697=1068.420,341.815,399.051,174.587,32.749,155.995
C08698=1068.427,342.063,399.016,174.591,32.755,155.996
C08699=1068.433,342.310,398.981,174.594,32.759,155.997
C08700=1068.439,342.557,398.946,174.598,32.765,155.998
C08701=1068.446,342.804,398.911,174.601,32.770,155.999
C08702=1068.452,343.052,398.875,174.605,32.775,156.000
C08703=1068.459,343.299,398.840,174.609,32.781,156.001
C08704=1068.465,343.547,398.805,174.612,32.785,156.002
C08705=1068.471,343.794,398.769,174.616,32.791,156.003
C08706=1068.478,344.042,398.734,174.620,32.796,156.005
C08707=1068.484,344.290,398.698,174.623,32.801,156.006
C08708=1068.490,344.515,398.665,174.627,32.806,156.007
C08709=1068.496,344.741,398.633,174.630,32.811,156.007
C08710=1068.502,344.966,398.601,174.633,32.816,156.008
C08711=1068.508,345.192,398.568,174.637,32.821,156.009
C08712=1068.514,345.418,398.536,174.640,32.826,156.010
C08713=1068.520,345.644,398.504,174.643,32.830,156.011
C08714=1068.525,345.870,398.470,174.647,32.835,156.012
C08715=1068.531,346.096,398.438,174.650,32.840,156.013
C08716=1068.538,346.343,398.403,174.654,32.845,156.014
C08717=1068.544,346.590,398.367,174.657,32.851,156.016
C08718=1068.551,346.838,398.331,174.661,32.856,156.017
C08719=1068.557,347.085,398.296,174.665,32.862,156.018
C08720=1068.564,347.332,398.259,174.668,32.867,156.019
C08721=1068.570,347.580,398.224,174.672,32.872,156.020
C08722=1068.576,347.827,398.189,174.676,32.877,156.021
C08723=1068.583,348.074,398.152,174.680,32.883,156.022
C08724=1068.590,348.322,398.117,174.683,32.888,156.023
C08725=1068.596,348.569,398.081,174.687,32.894,156.024
C08726=1068.602,348.816,398.045,174.691,32.899,156.025
C08727=1068.609,349.064,398.010,174.694,32.904,156.026
C08728=1068.615,349.311,397.973,174.698,32.910,156.027
C08729=1068.622,349.559,397.937,174.702,32.915,156.028
C08730=1068.629,349.806,397.901,174.706,32.921,156.030
C08731=1068.635,350.054,397.866,174.709,32.926,156.031
C08732=1068.641,350.301,397.829,174.713,32.931,156.032
C08733=1068.648,350.547,397.793,174.717,32.937,156.033
C08734=1068.654,350.795,397.757,174.721,32.943,156.034
C08735=1068.661,351.042,397.721,174.724,32.948,156.035
C08736=1068.667,351.290,397.684,174.728,32.953,156.036
C08737=1068.674,351.537,397.649,174.732,32.959,156.037
C08738=1068.681,351.784,397.613,174.736,32.964,156.038
C08739=1068.687,352.031,397.576,174.739,32.970,156.040
C08740=1068.693,352.279,397.540,174.743,32.975,156.041
C08741=1068.699,352.526,397.504,174.747,32.981,156.042
C08742=1068.707,352.773,397.468,174.751,32.986,156.043
C08743=1068.713,353.021,397.431,174.754,32.992,156.044
C08744=1068.719,353.268,397.396,174.758,32.998,156.045
C08745=1068.726,353.515,397.359,174.762,33.003,156.046
C08746=1068.732,353.762,397.323,174.766,33.009,156.047
C08747=1068.739,354.010,397.286,174.770,33.015,156.049
C08748=1068.745,354.257,397.249,174.773,33.020,156.050
C08749=1068.752,354.504,397.213,174.777,33.026,156.051
C08750=1068.758,354.751,397.177,174.781,33.031,156.052
C08751=1068.765,354.999,397.140,174.785,33.037,156.053
C08752=1068.771,355.246,397.103,174.789,33.043,156.054
C08753=1068.778,355.493,397.067,174.793,33.048,156.056
C08754=1068.784,355.740,397.030,174.797,33.054,156.057
C08755=1068.791,355.988,396.994,174.801,33.060,156.058
C08756=1068.797,356.235,396.957,174.805,33.065,156.059
C08757=1068.803,356.482,396.921,174.809,33.071,156.060
C08758=1068.810,356.730,396.884,174.813,33.077,156.061
C08759=1068.817,356.977,396.848,174.816,33.083,156.063
C08760=1068.823,357.224,396.811,174.820,33.088,156.064
C08761=1068.830,357.471,396.774,174.824,33.094,156.065
C08762=1068.837,357.718,396.737,174.828,33.100,156.066
C08763=1068.843,357.965,396.701,174.832,33.105,156.067
C08764=1068.850,358.193,396.667,174.835,33.111,156.068
C08765=1068.856,358.421,396.633,174.839,33.116,156.069
C08766=1068.862,358.648,396.599,174.842,33.121,156.071
C08767=1068.868,358.876,396.565,174.846,33.127,156.072
C08768=1068.874,359.104,396.532,174.850,33.132,156.073
C08769=1068.880,359.331,396.497,174.853,33.137,156.074
C08770=1068.886,359.559,396.463,174.857,33.143,156.075
C08771=1068.893,359.787,396.429,174.860,33.148,156.076
C08772=1068.898,360.034,396.392,174.864,33.154,156.077
C08773=1068.905,360.281,396.355,174.868,33.160,156.079
C08774=1068.912,360.528,396.318,174.873,33.166,156.080
C08775=1068.918,360.775,396.281,174.877,33.172,156.081
C08776=1068.926,361.022,396.244,174.881,33.177,156.082
C08777=1068.931,361.270,396.207,174.885,33.184,156.084
C08778=1068.938,361.517,396.169,174.889,33.189,156.085
C08779=1068.945,361.764,396.133,174.893,33.195,156.086
C08780=1068.952,362.011,396.095,174.896,33.201,156.087
C08781=1068.958,362.258,396.059,174.900,33.207,156.088
C08782=1068.965,362.505,396.021,174.904,33.213,156.090
C08783=1068.971,362.753,395.984,174.908,33.219,156.091
C08784=1068.978,363.000,395.947,174.912,33.225,156.092
C08785=1068.985,363.246,395.909,174.916,33.231,156.093
C08786=1068.992,363.494,395.871,174.920,33.237,156.095
C08787=1068.998,363.741,395.835,174.924,33.243,156.096
C08788=1069.005,363.988,395.797,174.929,33.249,156.097
C08789=1069.012,364.235,395.759,174.933,33.255,156.098
C08790=1069.018,364.482,395.723,174.937,33.261,156.100
C08791=1069.025,364.729,395.685,174.941,33.267,156.101
C08792=1069.031,364.976,395.648,174.945,33.273,156.102
C08793=1069.038,365.223,395.610,174.949,33.280,156.103
C08794=1069.044,365.470,395.572,174.953,33.285,156.105
C08795=1069.052,365.717,395.535,174.957,33.292,156.106
C08796=1069.058,365.965,395.497,174.961,33.298,156.107
C08797=1069.065,366.211,395.459,174.965,33.304,156.109
C08798=1069.071,366.458,395.421,174.970,33.310,156.110
C08799=1069.077,366.705,395.384,174.974,33.316,156.111
C08800=1069.084,366.952,395.346,174.978,33.323,156.113
C08801=1069.091,367.200,395.308,174.982,33.329,156.114
C08802=1069.098,367.446,395.271,174.986,33.335,156.115
C08803=1069.104,367.694,395.233,174.990,33.341,156.116
C08804=1069.111,367.941,395.195,174.994,33.347,156.118
C08805=1069.117,368.188,395.157,174.998,33.354,156.119
C08806=1069.124,368.435,395.120,175.002,33.360,156.120
C08807=1069.131,368.682,395.082,175.007,33.366,156.122
C08808=1069.138,368.928,395.044,175.011,33.373,156.123
C08809=1069.144,369.175,395.006,175.015,33.379,156.124
C08810=1069.151,369.423,394.968,175.019,33.385,156.126
C08811=1069.158,369.670,394.930,175.023,33.392,156.127
C08812=1069.164,369.916,394.892,175.027,33.398,156.128
C08813=1069.172,370.163,394.854,175.031,33.404,156.130
C08814=1069.178,370.411,394.816,175.035,33.410,156.131
C08815=1069.185,370.657,394.777,175.040,33.417,156.132
C08816=1069.192,370.904,394.740,175.044,33.423,156.134
C08817=1069.198,371.151,394.702,175.048,33.429,156.135
C08818=1069.206,371.398,394.664,175.052,33.436,156.136
C08819=1069.212,371.645,394.625,175.057,33.443,156.138
C08820=1069.218,371.881,394.589,175.060,33.448,156.139
C08821=1069.225,372.118,394.552,175.064,33.454,156.140
C08822=1069.232,372.353,394.516,175.069,33.461,156.142
C08823=1069.238,372.590,394.479,175.073,33.467,156.143
C08824=1069.244,372.826,394.442,175.077,33.473,156.144
C08825=1069.252,373.063,394.406,175.081,33.479,156.146
C08826=1069.258,373.299,394.369,175.085,33.485,156.147
C08827=1069.264,373.535,394.332,175.089,33.492,156.148
C08828=1069.272,373.782,394.294,175.093,33.498,156.150
C08829=1069.278,374.029,394.256,175.098,33.505,156.151
C08830=1069.284,374.275,394.217,175.102,33.512,156.153
C08831=1069.291,374.522,394.178,175.106,33.518,156.154
C08832=1069.298,374.769,394.139,175.111,33.525,156.155
C08833=1069.304,375.017,394.101,175.115,33.531,156.157
C08834=1069.311,375.263,394.062,175.119,33.538,156.158
C08835=1069.318,375.510,394.024,175.124,33.545,156.160
C08836=1069.325,375.757,393.985,175.128,33.551,156.161
C08837=1069.332,376.004,393.946,175.132,33.558,156.163
C08838=1069.339,376.251,393.907,175.136,33.564,156.164
C08839=1069.345,376.497,393.868,175.141,33.571,156.165
C08840=1069.352,376.745,393.830,175.146,33.578,156.167
C08841=1069.359,376.992,393.791,175.150,33.585,156.168
C08842=1069.365,377.239,393.752,175.154,33.592,156.170
C08843=1069.373,377.485,393.714,175.158,33.598,156.171
C08844=1069.380,377.732,393.675,175.163,33.605,156.173
C08845=1069.387,377.978,393.636,175.168,33.612,156.174
C08846=1069.394,378.225,393.597,175.172,33.619,156.176
C08847=1069.401,378.472,393.558,175.176,33.626,156.177
C08848=1069.407,378.719,393.519,175.180,33.632,156.179
C08849=1069.414,378.965,393.480,175.185,33.639,156.180
C08850=1069.421,379.212,393.442,175.190,33.646,156.182
C08851=1069.428,379.459,393.403,175.194,33.653,156.183
C08852=1069.435,379.705,393.363,175.198,33.660,156.184
C08853=1069.442,379.952,393.324,175.203,33.667,156.186
C08854=1069.449,380.200,393.285,175.207,33.673,156.187
C08855=1069.456,380.446,393.246,175.212,33.681,156.189
C08856=1069.463,380.693,393.207,175.216,33.687,156.191
C08857=1069.469,380.940,393.167,175.221,33.694,156.192
C08858=1069.476,381.187,393.129,175.225,33.701,156.193
C08859=1069.484,381.434,393.089,175.230,33.708,156.195
C08860=1069.491,381.680,393.050,175.234,33.715,156.197
C08861=1069.498,381.927,393.010,175.239,33.722,156.198
C08862=1069.504,382.174,392.971,175.243,33.729,156.200
C08863=1069.511,382.420,392.931,175.247,33.736,156.201
C08864=1069.518,382.667,392.892,175.253,33.744,156.203
C08865=1069.525,382.913,392.853,175.257,33.751,156.204
C08866=1069.531,383.161,392.813,175.261,33.758,156.206
C08867=1069.539,383.407,392.773,175.266,33.765,156.207
C08868=1069.546,383.653,392.734,175.271,33.772,156.209
C08869=1069.552,383.900,392.694,175.275,33.779,156.211
C08870=1069.559,384.147,392.655,175.279,33.787,156.212
C08871=1069.566,384.394,392.614,175.285,33.794,156.214
C08872=1069.573,384.641,392.576,175.289,33.801,156.215
C08873=1069.580,384.887,392.536,175.293,33.808,156.217
C08874=1069.587,385.134,392.496,175.298,33.815,156.218
C08875=1069.594,385.380,392.456,175.303,33.823,156.220
C08876=1069.601,385.636,392.415,175.308,33.830,156.222
C08877=1069.608,385.892,392.374,175.312,33.838,156.223
C08878=1069.615,386.147,392.332,175.318,33.846,156.225
C08879=1069.623,386.403,392.291,175.322,33.853,156.227
C08880=1069.630,386.649,392.251,175.327,33.861,156.228
C08881=1069.637,386.896,392.212,175.331,33.868,156.230
C08882=1069.644,387.143,392.171,175.336,33.875,156.232
C08883=1069.651,387.389,392.132,175.341,33.883,156.233
C08884=1069.658,387.635,392.092,175.345,33.890,156.235
C08885=1069.665,387.883,392.052,175.351,33.897,156.236
C08886=1069.672,388.129,392.012,175.355,33.905,156.238
C08887=1069.679,388.376,391.972,175.359,33.912,156.240
C08888=1069.686,388.622,391.932,175.365,33.919,156.241
C08889=1069.694,388.869,391.891,175.369,33.927,156.243
C08890=1069.701,389.115,391.851,175.374,33.935,156.245
C08891=1069.708,389.362,391.811,175.378,33.942,156.246
C08892=1069.715,389.608,391.771,175.384,33.950,156.248
C08893=1069.723,389.855,391.730,175.388,33.957,156.250
C08894=1069.729,390.101,391.690,175.393,33.965,156.251
C08895=1069.737,390.348,391.650,175.398,33.973,156.253
C08896=1069.743,390.595,391.610,175.403,33.980,156.255
C08897=1069.751,390.841,391.570,175.407,33.988,156.257
C08898=1069.758,391.088,391.529,175.413,33.995,156.258
C08899=1069.765,391.334,391.488,175.417,34.003,156.260
C08900=1069.773,391.581,391.448,175.423,34.010,156.262
C08901=1069.779,391.827,391.407,175.427,34.018,156.263
C08902=1069.786,392.074,391.367,175.432,34.026,156.265
C08903=1069.794,392.320,391.327,175.437,34.034,156.267
C08904=1069.801,392.567,391.286,175.442,34.042,156.269
C08905=1069.808,392.813,391.245,175.446,34.049,156.270
C08906=1069.814,393.060,391.205,175.452,34.057,156.272
C08907=1069.822,393.306,391.164,175.456,34.065,156.274
C08908=1069.830,393.553,391.123,175.462,34.073,156.276
C08909=1069.836,393.799,391.083,175.466,34.081,156.277
C08910=1069.843,394.046,391.042,175.471,34.089,156.279
C08911=1069.851,394.292,391.001,175.476,34.097,156.281
C08912=1069.858,394.538,390.960,175.481,34.105,156.283
C08913=1069.865,394.785,390.920,175.485,34.113,156.285
C08914=1069.872,395.032,390.878,175.491,34.121,156.286
C08915=1069.880,395.278,390.837,175.496,34.129,156.288
C08916=1069.886,395.524,390.796,175.501,34.137,156.290
C08917=1069.894,395.771,390.755,175.506,34.145,156.292
C08918=1069.901,396.018,390.714,175.511,34.153,156.294
C08919=1069.909,396.264,390.673,175.516,34.161,156.295
C08920=1069.916,396.510,390.632,175.521,34.169,156.297
C08921=1069.923,396.756,390.591,175.526,34.177,156.299
C08922=1069.930,397.003,390.550,175.531,34.185,156.301
C08923=1069.938,397.249,390.509,175.536,34.193,156.303
C08924=1069.945,397.496,390.467,175.541,34.202,156.305
C08925=1069.952,397.743,390.426,175.547,34.210,156.306
C08926=1069.959,397.989,390.385,175.551,34.218,156.308
C08927=1069.967,398.236,390.344,175.556,34.227,156.310
C08928=1069.974,398.482,390.302,175.562,34.235,156.312
C08929=1069.981,398.728,390.261,175.566,34.243,156.314
C08930=1069.988,398.974,390.220,175.572,34.251,156.316
C08931=1069.995,399.221,390.178,175.577,34.260,156.318
C08932=1070.003,399.493,390.132,175.583,34.269,156.320
C08933=1070.011,399.764,390.086,175.588,34.278,156.322
C08934=1070.019,400.036,390.040,175.594,34.287,156.324
C08935=1070.028,400.307,389.994,175.599,34.297,156.326
C08936=1070.035,400.554,389.953,175.605,34.305,156.328
C08937=1070.042,400.800,389.911,175.610,34.314,156.330
C08938=1070.050,401.046,389.870,175.615,34.322,156.332
C08939=1070.057,401.292,389.828,175.620,34.331,156.334
C08940=1070.065,401.539,389.787,175.626,34.339,156.336
C08941=1070.071,401.785,389.744,175.631,34.348,156.338
C08942=1070.079,402.032,389.703,175.636,34.356,156.340
C08943=1070.086,402.278,389.661,175.642,34.365,156.342
C08944=1070.094,402.524,389.619,175.647,34.373,156.344
C08945=1070.101,402.770,389.578,175.653,34.382,156.346
C08946=1070.109,403.017,389.535,175.657,34.391,156.348
C08947=1070.116,403.263,389.493,175.663,34.400,156.350
C08948=1070.124,403.509,389.451,175.668,34.408,156.352
C08949=1070.130,403.756,389.409,175.674,34.417,156.354
C08950=1070.138,404.002,389.367,175.679,34.426,156.356
C08951=1070.146,404.248,389.325,175.684,34.435,156.358
C08952=1070.153,404.495,389.282,175.689,34.444,156.360
C08953=1070.161,404.741,389.240,175.695,34.452,156.362
C08954=1070.168,404.987,389.198,175.701,34.461,156.364
C08955=1070.175,405.233,389.156,175.706,34.470,156.366
C08956=1070.183,405.480,389.113,175.712,34.479,156.368
C08957=1070.190,405.726,389.071,175.717,34.488,156.370
C08958=1070.198,405.972,389.029,175.722,34.497,156.372
C08959=1070.205,406.219,388.986,175.728,34.506,156.374
C08960=1070.213,406.465,388.944,175.733,34.515,156.376
C08961=1070.220,406.712,388.902,175.739,34.524,156.379
C08962=1070.227,406.958,388.860,175.744,34.533,156.381
C08963=1070.235,407.204,388.816,175.750,34.542,156.383
C08964=1070.242,407.450,388.774,175.756,34.552,156.385
C08965=1070.249,407.696,388.732,175.761,34.561,156.387
C08966=1070.257,407.943,388.688,175.767,34.570,156.389
C08967=1070.264,408.189,388.645,175.773,34.579,156.391
C08968=1070.272,408.436,388.603,175.778,34.589,156.394
C08969=1070.279,408.681,388.560,175.784,34.598,156.396
C08970=1070.286,408.928,388.517,175.790,34.607,156.398
C08971=1070.295,409.174,388.474,175.795,34.616,156.400
C08972=1070.302,409.420,388.432,175.801,34.626,156.402
C08973=1070.309,409.666,388.388,175.807,34.635,156.404
C08974=1070.317,409.912,388.346,175.812,34.645,156.407
C08975=1070.325,410.159,388.303,175.818,34.654,156.409
C08976=1070.332,410.405,388.260,175.824,34.663,156.411
C08977=1070.340,410.651,388.217,175.829,34.673,156.413
C08978=1070.347,410.897,388.174,175.835,34.682,156.415
C08979=1070.355,411.144,388.131,175.841,34.692,156.418
C08980=1070.363,411.390,388.088,175.847,34.701,156.420
C08981=1070.370,411.635,388.045,175.852,34.711,156.422
C08982=1070.378,411.882,388.001,175.858,34.720,156.424
C08983=1070.385,412.127,387.958,175.864,34.730,156.427
C08984=1070.394,412.374,387.915,175.869,34.739,156.429
C08985=1070.401,412.620,387.872,175.875,34.749,156.431
C08986=1070.408,412.866,387.828,175.881,34.759,156.433
C08987=1070.416,413.112,387.785,175.888,34.769,156.436
C08988=1070.430,413.527,387.712,175.897,34.785,156.440
C08989=1070.443,413.942,387.639,175.907,34.802,156.444
C08990=1070.456,414.356,387.565,175.918,34.818,156.448
C08991=1070.469,414.771,387.492,175.928,34.834,156.451
C08992=1070.477,415.018,387.448,175.934,34.845,156.454
C08993=1070.485,415.264,387.404,175.940,34.854,156.456
C08994=1070.492,415.509,387.361,175.945,34.865,156.459
C08995=1070.500,415.755,387.317,175.951,34.875,156.461
C08996=1070.508,416.002,387.273,175.958,34.885,156.463
C08997=1070.516,416.248,387.229,175.964,34.895,156.466
C08998=1070.524,416.494,387.185,175.970,34.905,156.468
C08999=1070.531,416.739,387.141,175.976,34.915,156.471
C09000=1070.539,416.985,387.098,175.983,34.925,156.473
C09001=1070.547,417.231,387.053,175.988,34.936,156.475
C09002=1070.554,417.478,387.009,175.994,34.946,156.478
C09003=1070.562,417.724,386.965,176.001,34.956,156.480
C09004=1070.570,417.969,386.921,176.007,34.966,156.483
C09005=1070.578,418.216,386.877,176.013,34.977,156.485
C09006=1070.586,418.461,386.833,176.020,34.987,156.488
C09007=1070.594,418.707,386.788,176.026,34.997,156.490
C09008=1070.602,418.953,386.745,176.032,35.008,156.493
C09009=1070.610,419.199,386.700,176.039,35.018,156.495
C09010=1070.617,419.445,386.655,176.045,35.029,156.498
C09011=1070.625,419.691,386.611,176.052,35.040,156.500
C09012=1070.633,419.937,386.567,176.058,35.050,156.503
C09013=1070.641,420.183,386.522,176.065,35.060,156.505
C09014=1070.649,420.428,386.478,176.071,35.071,156.508
C09015=1070.657,420.674,386.434,176.077,35.082,156.511
C09016=1070.665,420.920,386.389,176.083,35.092,156.513
C09017=1070.673,421.167,386.344,176.089,35.103,156.516
C09018=1070.682,421.412,386.300,176.097,35.114,156.518
C09019=1070.689,421.658,386.255,176.103,35.125,156.521
C09020=1070.697,421.904,386.210,176.110,35.135,156.523
C09021=1070.705,422.150,386.166,176.116,35.146,156.526
C09022=1070.713,422.395,386.120,176.123,35.157,156.529
C09023=1070.721,422.641,386.076,176.129,35.168,156.531
C09024=1070.729,422.888,386.031,176.136,35.179,156.534
C09025=1070.737,423.133,385.986,176.143,35.190,156.537
C09026=1070.744,423.379,385.941,176.149,35.201,156.539
C09027=1070.753,423.624,385.896,176.156,35.212,156.542
C09028=1070.765,423.977,385.831,176.165,35.228,156.546
C09029=1070.776,424.329,385.767,176.175,35.244,156.550
C09030=1070.788,424.681,385.702,176.185,35.260,156.554
C09031=1070.800,425.033,385.637,176.194,35.276,156.558
C09032=1070.807,425.279,385.592,176.201,35.287,156.560
C09033=1070.816,425.524,385.547,176.208,35.298,156.563
C09034=1070.824,425.771,385.501,176.215,35.310,156.566
C09035=1070.832,426.016,385.456,176.222,35.321,156.569
C09036=1070.840,426.262,385.410,176.228,35.332,156.572
C09037=1070.849,426.507,385.365,176.235,35.343,156.574
C09038=1070.857,426.753,385.319,176.242,35.355,156.577
C09039=1070.865,426.999,385.274,176.250,35.367,156.580
C09040=1070.875,427.293,385.220,176.257,35.380,156.583
C09041=1070.885,427.587,385.164,176.266,35.394,156.587
C09042=1070.894,427.881,385.109,176.274,35.408,156.590
C09043=1070.904,428.175,385.055,176.283,35.422,156.594
C09044=1070.912,428.420,385.010,176.290,35.434,156.597
C09045=1070.921,428.666,384.964,176.297,35.445,156.599
C09046=1070.929,428.912,384.918,176.304,35.458,156.602
C09047=1070.937,429.157,384.872,176.311,35.469,156.605
C09048=1070.945,429.403,384.825,176.318,35.481,156.608
C09049=1070.954,429.648,384.780,176.325,35.493,156.611
C09050=1070.962,429.894,384.734,176.333,35.505,156.614
C09051=1070.971,430.140,384.687,176.340,35.517,156.617
C09052=1070.978,430.385,384.642,176.347,35.529,156.620
C09053=1070.987,430.630,384.595,176.355,35.541,156.623
C09054=1070.996,430.876,384.549,176.362,35.553,156.626
C09055=1071.004,431.122,384.503,176.369,35.565,156.629
C09056=1071.012,431.367,384.457,176.377,35.577,156.632
C09057=1071.020,431.613,384.411,176.384,35.589,156.635
C09058=1071.029,431.858,384.364,176.392,35.602,156.638
C09059=1071.038,432.104,384.317,176.399,35.614,156.641
C09060=1071.045,432.349,384.271,176.406,35.626,156.644
C09061=1071.054,432.594,384.224,176.414,35.638,156.647
C09062=1071.063,432.840,384.177,176.421,35.651,156.651
C09063=1071.071,433.085,384.131,176.429,35.664,156.654
C09064=1071.080,433.331,384.084,176.436,35.676,156.657
C09065=1071.088,433.576,384.037,176.444,35.689,156.660
C09066=1071.096,433.821,383.991,176.451,35.701,156.663
C09067=1071.105,434.066,383.944,176.459,35.714,156.666
C09068=1071.113,434.312,383.897,176.466,35.726,156.670
C09069=1071.121,434.558,383.850,176.474,35.739,156.673
C09070=1071.130,434.803,383.802,176.481,35.752,156.676
C09071=1071.138,435.048,383.756,176.490,35.765,156.679
C09072=1071.147,435.294,383.709,176.498,35.778,156.682
C09073=1071.156,435.539,383.662,176.505,35.790,156.686
C09074=1071.164,435.784,383.615,176.513,35.803,156.689
C09075=1071.173,436.030,383.568,176.520,35.816,156.692
C09076=1071.182,436.275,383.521,176.529,35.829,156.696
C09077=1071.190,436.520,383.474,176.537,35.842,156.699
C09078=1071.199,436.766,383.426,176.544,35.855,156.702
C09079=1071.208,437.011,383.378,176.552,35.868,156.705
C09080=1071.216,437.256,383.331,176.561,35.881,156.709
C09081=1071.225,437.501,383.284,176.568,35.894,156.712
C09082=1071.234,437.746,383.236,176.576,35.908,156.716
C09083=1071.243,437.991,383.189,176.585,35.921,156.719
C09084=1071.251,438.238,383.141,176.593,35.934,156.722
C09085=1071.260,438.482,383.094,176.600,35.947,156.726
C09086=1071.269,438.727,383.046,176.609,35.961,156.729
C09087=1071.279,438.973,382.999,176.617,35.974,156.733
C09088=1071.287,439.218,382.951,176.626,35.988,156.736
C09089=1071.296,439.463,382.903,176.633,36.001,156.739
C09090=1071.304,439.709,382.855,176.641,36.015,156.743
C09091=1071.313,439.954,382.807,176.650,36.029,156.747
C09092=1071.322,440.198,382.759,176.658,36.042,156.750
C09093=1071.331,440.444,382.711,176.667,36.056,156.754
C09094=1071.340,440.689,382.663,176.675,36.069,156.757
C09095=1071.348,440.933,382.615,176.684,36.083,156.761
C09096=1071.358,441.193,382.563,176.693,36.098,156.764
C09097=1071.367,441.451,382.513,176.702,36.113,156.768
C09098=1071.376,441.709,382.462,176.711,36.127,156.772
C09099=1071.386,441.968,382.411,176.720,36.142,156.776
C09100=1071.395,442.213,382.363,176.728,36.156,156.779
C09101=1071.404,442.459,382.314,176.737,36.170,156.783
C09102=1071.413,442.703,382.266,176.745,36.184,156.787
C09103=1071.422,442.949,382.218,176.754,36.199,156.791
C09104=1071.431,443.193,382.169,176.763,36.213,156.794
C09105=1071.440,443.438,382.120,176.771,36.227,156.798
C09106=1071.449,443.684,382.071,176.780,36.241,156.802
